IF st_config_achse.b_config_fertig THEN
	(* Fehlermeldungen und Betriebsmeldungen ab dem Startindex in die globalen Meldungsarrays schreiben *)
	garr_stoermeldungen[st_config_achse.i16_meld_startindex + 0] := st_sm.b_achse_nicht_bb;
	garr_stoermeldungen[st_config_achse.i16_meld_startindex + 1] := st_sm.b_achse_nicht_referenziert;
	garr_stoermeldungen[st_config_achse.i16_meld_startindex + 2] := st_sm.b_keine_verfahrfreigabe;
	garr_stoermeldungen[st_config_achse.i16_meld_startindex + 3] := st_sm.b_achse_nicht_auf_startpos;
	garr_stoermeldungen[st_config_achse.i16_meld_startindex + 4] := st_sm.b_ende_skalierungs_nocke;
	garr_stoermeldungen[st_config_achse.i16_meld_startindex + 5] := st_sm.b_ende_camming_nocke;
	garr_stoermeldungen[st_config_achse.i16_meld_startindex + 6] := st_sm.b_skalierung_noch_aktiv;
	garr_stoermeldungen[st_config_achse.i16_meld_startindex + 7] := FALSE;
	garr_stoermeldungen[st_config_achse.i16_meld_startindex + 8] := FALSE;
	garr_stoermeldungen[st_config_achse.i16_meld_startindex + 9] := FALSE;
	garr_stoermeldungen[st_config_achse.i16_meld_startindex + 10] := sm_kein_nocken_definiert;
	garr_stoermeldungen[st_config_achse.i16_meld_startindex + 11] := FALSE;
	garr_stoermeldungen[st_config_achse.i16_meld_startindex + 12] := FALSE;
	garr_stoermeldungen[st_config_achse.i16_meld_startindex + 13] := FALSE;
	garr_stoermeldungen[st_config_achse.i16_meld_startindex + 14] := FALSE;
	garr_stoermeldungen[st_config_achse.i16_meld_startindex + 15] := FALSE;
	garr_stoermeldungen[st_config_achse.i16_meld_startindex + 16] := st_drive_cmd.meldungen.sm_write_soe_parameter;
	garr_stoermeldungen[st_config_achse.i16_meld_startindex + 17] := st_drive_cmd.meldungen.sm_read_soe_parameter;
	garr_stoermeldungen[st_config_achse.i16_meld_startindex + 18] := st_drive_cmd.meldungen.sm_write_nc_parameter;
	garr_stoermeldungen[st_config_achse.i16_meld_startindex + 19] := st_drive_cmd.meldungen.sm_read_nc_parameter;
	garr_stoermeldungen[st_config_achse.i16_meld_startindex + 20] := st_drive_cmd.meldungen.sm_power_enable;
	garr_stoermeldungen[st_config_achse.i16_meld_startindex + 21] := st_drive_cmd.meldungen.sm_power_disable;
	garr_stoermeldungen[st_config_achse.i16_meld_startindex + 22] := st_drive_cmd.meldungen.sm_reset;
	garr_stoermeldungen[st_config_achse.i16_meld_startindex + 23] := st_drive_cmd.meldungen.sm_home;
	garr_stoermeldungen[st_config_achse.i16_meld_startindex + 24] := st_drive_cmd.meldungen.sm_setposition;
	garr_stoermeldungen[st_config_achse.i16_meld_startindex + 25] := st_drive_cmd.meldungen.sm_jog_vorwaerts;
	garr_stoermeldungen[st_config_achse.i16_meld_startindex + 26] := st_drive_cmd.meldungen.sm_jog_rueckwaerts;
	garr_stoermeldungen[st_config_achse.i16_meld_startindex + 27] := st_drive_cmd.meldungen.sm_move_absolute;
	garr_stoermeldungen[st_config_achse.i16_meld_startindex + 28] := st_drive_cmd.meldungen.sm_move_relative;
	garr_stoermeldungen[st_config_achse.i16_meld_startindex + 29] := st_drive_cmd.meldungen.sm_move_velocity;
	garr_stoermeldungen[st_config_achse.i16_meld_startindex + 30] := st_drive_cmd.meldungen.sm_move_modulo;
	garr_stoermeldungen[st_config_achse.i16_meld_startindex + 31] := st_drive_cmd.meldungen.sm_stop_axis;
	garr_stoermeldungen[st_config_achse.i16_meld_startindex + 32] := st_drive_cmd.meldungen.sm_halt_axis;
	garr_stoermeldungen[st_config_achse.i16_meld_startindex + 33] := st_drive_cmd.meldungen.sm_motion_command_timeout;
	garr_stoermeldungen[st_config_achse.i16_meld_startindex + 34] := st_sm.b_achsfehler;
	garr_stoermeldungen[st_config_achse.i16_meld_startindex + 35] := st_sm.b_devicefehler;
	garr_stoermeldungen[st_config_achse.i16_meld_startindex + 36] := st_drive_cmd.meldungen.sm_limit_positiv_erreicht;
	garr_stoermeldungen[st_config_achse.i16_meld_startindex + 37] := st_drive_cmd.meldungen.sm_limit_negativ_erreicht;
	garr_stoermeldungen[st_config_achse.i16_meld_startindex + 38] := st_drive_cmd.meldungen.sm_ec_coe_sdo_write_ex;
	garr_stoermeldungen[st_config_achse.i16_meld_startindex + 39] := st_drive_cmd.meldungen.sm_ec_coe_sdo_read_ex;
	garr_stoermeldungen[st_config_achse.i16_meld_startindex + 40] := FALSE;
	garr_stoermeldungen[st_config_achse.i16_meld_startindex + 41] := FALSE;
	garr_stoermeldungen[st_config_achse.i16_meld_startindex + 42] := FALSE;
	garr_stoermeldungen[st_config_achse.i16_meld_startindex + 43] := FALSE;
	garr_stoermeldungen[st_config_achse.i16_meld_startindex + 44] := FALSE;
	garr_stoermeldungen[st_config_achse.i16_meld_startindex + 45] := FALSE;
	garr_stoermeldungen[st_config_achse.i16_meld_startindex + 46] := FALSE;
	garr_stoermeldungen[st_config_achse.i16_meld_startindex + 47] := FALSE;
	garr_stoermeldungen[st_config_achse.i16_meld_startindex + 48] := FALSE;
	garr_stoermeldungen[st_config_achse.i16_meld_startindex + 49] := FALSE;

	garr_betriebsmeldungen[st_config_achse.i16_meld_startindex + 0] := FALSE;
	garr_betriebsmeldungen[st_config_achse.i16_meld_startindex + 1] := FALSE;
	garr_betriebsmeldungen[st_config_achse.i16_meld_startindex + 2] := FALSE;
	garr_betriebsmeldungen[st_config_achse.i16_meld_startindex + 3] := FALSE;
	garr_betriebsmeldungen[st_config_achse.i16_meld_startindex + 4] := FALSE;
	garr_betriebsmeldungen[st_config_achse.i16_meld_startindex + 5] := FALSE;
	garr_betriebsmeldungen[st_config_achse.i16_meld_startindex + 6] := FALSE;
	garr_betriebsmeldungen[st_config_achse.i16_meld_startindex + 7] := FALSE;
	garr_betriebsmeldungen[st_config_achse.i16_meld_startindex + 8] := FALSE;
	garr_betriebsmeldungen[st_config_achse.i16_meld_startindex + 9] := FALSE;
	garr_betriebsmeldungen[st_config_achse.i16_meld_startindex + 10] := FALSE;
	garr_betriebsmeldungen[st_config_achse.i16_meld_startindex + 11] := FALSE;
	garr_betriebsmeldungen[st_config_achse.i16_meld_startindex + 12] := FALSE;
	garr_betriebsmeldungen[st_config_achse.i16_meld_startindex + 13] := FALSE;
	garr_betriebsmeldungen[st_config_achse.i16_meld_startindex + 14] := FALSE;
	garr_betriebsmeldungen[st_config_achse.i16_meld_startindex + 15] := FALSE;
	garr_betriebsmeldungen[st_config_achse.i16_meld_startindex + 16] := FALSE;
	garr_betriebsmeldungen[st_config_achse.i16_meld_startindex + 17] := FALSE;
	garr_betriebsmeldungen[st_config_achse.i16_meld_startindex + 18] := FALSE;
	garr_betriebsmeldungen[st_config_achse.i16_meld_startindex + 19] := FALSE;
	garr_betriebsmeldungen[st_config_achse.i16_meld_startindex + 20] := FALSE;
	garr_betriebsmeldungen[st_config_achse.i16_meld_startindex + 21] := FALSE;
	garr_betriebsmeldungen[st_config_achse.i16_meld_startindex + 22] := FALSE;
	garr_betriebsmeldungen[st_config_achse.i16_meld_startindex + 23] := FALSE;
	garr_betriebsmeldungen[st_config_achse.i16_meld_startindex + 24] := FALSE;
	garr_betriebsmeldungen[st_config_achse.i16_meld_startindex + 25] := FALSE;
	garr_betriebsmeldungen[st_config_achse.i16_meld_startindex + 26] := FALSE;
	garr_betriebsmeldungen[st_config_achse.i16_meld_startindex + 27] := FALSE;
	garr_betriebsmeldungen[st_config_achse.i16_meld_startindex + 28] := FALSE;
	garr_betriebsmeldungen[st_config_achse.i16_meld_startindex + 29] := FALSE;
	garr_betriebsmeldungen[st_config_achse.i16_meld_startindex + 30] := FALSE;
	garr_betriebsmeldungen[st_config_achse.i16_meld_startindex + 31] := FALSE;
	garr_betriebsmeldungen[st_config_achse.i16_meld_startindex + 32] := FALSE;
	garr_betriebsmeldungen[st_config_achse.i16_meld_startindex + 33] := FALSE;
	garr_betriebsmeldungen[st_config_achse.i16_meld_startindex + 34] := FALSE;
	garr_betriebsmeldungen[st_config_achse.i16_meld_startindex + 35] := FALSE;
	garr_betriebsmeldungen[st_config_achse.i16_meld_startindex + 36] := FALSE;
	garr_betriebsmeldungen[st_config_achse.i16_meld_startindex + 37] := FALSE;
	garr_betriebsmeldungen[st_config_achse.i16_meld_startindex + 38] := FALSE;
	garr_betriebsmeldungen[st_config_achse.i16_meld_startindex + 39] := FALSE;
	garr_betriebsmeldungen[st_config_achse.i16_meld_startindex + 40] := FALSE;
	garr_betriebsmeldungen[st_config_achse.i16_meld_startindex + 41] := FALSE;
	garr_betriebsmeldungen[st_config_achse.i16_meld_startindex + 42] := FALSE;
	garr_betriebsmeldungen[st_config_achse.i16_meld_startindex + 43] := FALSE;
	garr_betriebsmeldungen[st_config_achse.i16_meld_startindex + 44] := FALSE;
	garr_betriebsmeldungen[st_config_achse.i16_meld_startindex + 45] := FALSE;
	garr_betriebsmeldungen[st_config_achse.i16_meld_startindex + 46] := FALSE;
	garr_betriebsmeldungen[st_config_achse.i16_meld_startindex + 47] := FALSE;
	garr_betriebsmeldungen[st_config_achse.i16_meld_startindex + 48] := FALSE;
	garr_betriebsmeldungen[st_config_achse.i16_meld_startindex + 49] := FALSE;
END_IF
END_PROGRAM

(* POU Maschine1720/WT Transport/ST_WT_Transport_Warteposition_1720, ST *)
PROGRAM ST_WT_Transport_Warteposition_1720
VAR_INPUT
	st_config								: struct_config;
	st_ctrl_in								: struct_ctrl_in;
	e_station_vorher_in_anforderung			: BOOL := FALSE;
	e_station_vorher_in_abgegeben			: BOOL := FALSE;
END_VAR
VAR_IN_OUT
	st_visu								: struct_visu;
END_VAR
VAR_OUTPUT
	st_ctrl_out							: struct_ctrl_out;
	a_station_vorher_out_erlaubnis			: BOOL := FALSE;
	a_station_vorher_out_angekommen		: BOOL := FALSE;
END_VAR
VAR
	fb_ton_uez							: TON;
	fb_ton_wz							: TON;
	fb_ton_quitt							: TON;
	fb_ton_wt_auf_wartepos				: TON;
	fb_tof_wt_auf_wartepos					: TOF;
	fb_r_trig_start							: R_TRIG;
	fb_r_trig_wartepos						: R_TRIG;
	fb_r_trig_wartepos_verlassen			: R_TRIG;
	fb_state_entry							: ST_StateEntry;
	sm_wt_hat_wartepos_nicht_verlassen	: BOOL := FALSE;
	sm_wt_hat_wartepos_ueberfahren		: BOOL := FALSE;
	bm_warte_anforderung					: BOOL := FALSE;
	bm_warte_wt_an_stopper				: BOOL := FALSE;
	bm_warte_beladepos_frei				: BOOL := FALSE;

	e_wt_auf_wartepos					AT %I* : BOOL;
	e_wt_wartepos_verlassen				AT %I* : BOOL;
END_VAR
(* Zeiten *)
fb_ton_uez(IN:= , PT:= , Q=>  , ET=> );
fb_ton_wz(IN:= , PT:= , Q=> , ET=> );
fb_ton_quitt(IN:= , PT:= t#100ms, Q=> , ET=> );

fb_ton_wt_auf_wartepos(IN:= e_wt_auf_wartepos, PT:= t#200ms, Q=> , ET=> );
fb_tof_wt_auf_wartepos(IN:= e_wt_auf_wartepos, PT:= t#200ms, Q=> , ET=> );

(* Flanken *)
fb_r_trig_wartepos(CLK:= e_wt_auf_wartepos, Q=> );
fb_r_trig_wartepos_verlassen(CLK:= e_wt_wartepos_verlassen, Q=> );
fb_r_trig_start(CLK:= st_ctrl_in.b_start, Q=> );

(* ==================================Toplevel=================================== *)
IF fb_state_entry.i16_next_step > INIT AND fb_state_entry.i16_next_step < FEHLER THEN
	(* Allgemeine Fehler *)
	IF st_ctrl_in.b_stop THEN
		fb_state_entry.i16_next_step := STOP;
	ELSIF zyl_wt_stopper_einlauf.st_ctrl.out.b_fehler THEN
		fb_state_entry.i16_next_step := FEHLER;
	(* Zylinder im Handbetrieb *)
	ELSIF gi16_betriebsart = HAND AND
		st_visu.st_zyl.i16_nr_zyl_im_handbetrieb = zyl_wt_stopper_einlauf.fb.st_config.i16_identnummer
		THEN
			fb_state_entry.i16_next_step := FEHLER;
	END_IF
END_IF

(* ============================Haupt-Schrittkette================================ *)
fb_state_entry(
	i16_next_step:= , 
	i16_pos:= 1,
	s_debugtext:= ,
	E=> ,
	X=> , 
	i16_step=> ,
	i16_last_step=> );

CASE fb_state_entry.i16_step OF
(*=======================================================*)
	INIT_OBJ:
		IF st_config.b_config_fertig THEN
			fb_state_entry.i16_next_step := INIT;
		END_IF

(*=======================================================*)
	INIT:
		IF fb_state_entry.E THEN
			fb_ton_wz.IN := FALSE;
			fb_ton_uez.IN := FALSE;
			fb_ton_quitt.IN := FALSE;
			st_ctrl_out.b_fehler := FALSE;
			st_ctrl_out.b_bereit := FALSE;
			st_ctrl_out.b_fertig := FALSE;
			st_ctrl_out.b_kontroller_start := FALSE;
			zyl_wt_stopper_einlauf.st_ctrl.in.b_einfahren := FALSE;
			zyl_wt_stopper_einlauf.st_ctrl.in.b_ausfahren := FALSE;
			sm_wt_hat_wartepos_nicht_verlassen := FALSE;
			sm_wt_hat_wartepos_ueberfahren := FALSE;
			bm_warte_anforderung := FALSE;
			bm_warte_wt_an_stopper := FALSE;
			bm_warte_beladepos_frei := FALSE;
			a_station_vorher_out_erlaubnis := FALSE;
			a_station_vorher_out_angekommen := FALSE;
		END_IF

		(*-----------------------Weiterschaltbedingungen----------------------------*)
		IF st_ctrl_in.b_init THEN
			zyl_wt_stopper_einlauf.st_ctrl.in.b_quittieren := FALSE;
			fb_state_entry.i16_next_step := 20;
		END_IF

(*=======================================================*)
	20: (* Initialisierung: Einlaufstopper ausfahren *)
		IF fb_state_entry.E THEN
			zyl_wt_stopper_einlauf.st_ctrl.in.b_ausfahren := TRUE;
		END_IF

		(*-----------------------Weiterschaltbedingungen----------------------------*)
		IF zyl_wt_stopper_einlauf.st_ctrl.out.b_ausgefahren THEN
			zyl_wt_stopper_einlauf.st_ctrl.in.b_ausfahren := FALSE;
			fb_state_entry.i16_next_step :=  BEREIT;
		END_IF

(*=======================================================*)
	BEREIT:	(* Warte auf Start von Kontroller *)
		IF fb_state_entry.E THEN
			st_ctrl_out.b_bereit := TRUE;
			st_ctrl_out.b_fertig := TRUE;
		END_IF

	(*-----------------------Weiterschaltbedingungen----------------------------*)
		IF st_config.b_station_aktiv OR st_config.b_station_in_simulation THEN
			(* WT Transport aktiv oder in Simulation *)
			IF st_ctrl_in.b_start THEN
			(* WT Transport gestartet *)
				st_ctrl_out.b_fertig := FALSE;
				fb_state_entry.i16_next_step := 110;
			END_IF
		ELSE
			fb_state_entry.i16_next_step := 500;
		END_IF

(*=======================================================*)
	110: (* Statische WT-Abfrage auf Warteposition nach der Initialisierung *)
		IF fb_state_entry.E THEN
			st_ctrl_out.b_kontroller_start := TRUE;
		END_IF

		IF NOT e_station_vorher_in_abgegeben THEN
			a_station_vorher_out_angekommen := FALSE;
		END_IF

		(*-----------------------Weiterschaltbedingungen----------------------------*)
		IF e_wt_auf_wartepos THEN
			st_ctrl_out.b_kontroller_start := FALSE;
			fb_state_entry.i16_next_step := 140;
		ELSE	(* Kein WT da, deshalb einen holen *)
			st_ctrl_out.b_kontroller_start := FALSE;
			fb_state_entry.i16_next_step := 120;
		END_IF

(*=======================================================*)
	120: (* Kein WT da -> warte auf Anforderung von vorheriger Station *)
		IF fb_state_entry.E THEN
			st_ctrl_out.b_kontroller_start := TRUE;
			bm_warte_anforderung := TRUE;
		END_IF

		IF NOT e_station_vorher_in_abgegeben THEN
			a_station_vorher_out_angekommen := FALSE;
		END_IF

		(*-----------------------Weiterschaltbedingungen----------------------------*)
		IF e_station_vorher_in_anforderung THEN
			a_station_vorher_out_angekommen := FALSE;
			a_station_vorher_out_erlaubnis := TRUE;
			st_ctrl_out.b_kontroller_start := FALSE;
			bm_warte_anforderung := FALSE;
			fb_state_entry.i16_next_step := 130;
		END_IF

(*=======================================================*)
	130: (* Warte bis WT an Stopper angekommen ist *)
		IF fb_state_entry.E THEN
			st_ctrl_out.b_kontroller_start := TRUE;
			bm_warte_wt_an_stopper := TRUE;
		END_IF

		(*-----------------------Weiterschaltbedingungen----------------------------*)
		IF fb_r_trig_wartepos.Q THEN
			a_station_vorher_out_erlaubnis := FALSE;
			a_station_vorher_out_angekommen := TRUE;
			st_ctrl_out.b_kontroller_start := FALSE;
			fb_ton_uez.IN := FALSE;
			bm_warte_wt_an_stopper := FALSE;
			fb_state_entry.i16_next_step := 140;
		END_IF

(*=======================================================*)
	140: (* WT ist da - Warten bis Beladeposition auf Bestücktisch frei ist *)
		IF fb_state_entry.E THEN
			zyl_wt_stopper_einlauf.st_ctrl.in.b_ausfahren := FALSE;
			zyl_wt_stopper_einlauf.st_ctrl.in.b_einfahren := FALSE;
			bm_warte_beladepos_frei := TRUE;
		END_IF

		(*-----------------------Weiterschaltbedingungen----------------------------*)
		IF NOT ST_WT_Transport_Beladen_1720.e_wt_auf_beladepos AND NOT axis_z_achse.st_ctrl.in.b_start THEN
			bm_warte_beladepos_frei := FALSE;
			fb_state_entry.i16_next_step := 150;
		ELSIF e_wt_wartepos_verlassen THEN
			(* Warteposition wurde unerlaubterweise überfahren *)
			sm_wt_hat_wartepos_ueberfahren := TRUE;
			fb_state_entry.i16_next_step := FEHLER;
		END_IF

(*=======================================================*)
	150: (* Bestücktisch ist frei -> Einlaufstopper einfahren *)
		IF fb_state_entry.E THEN
			zyl_wt_stopper_einlauf.st_ctrl.in.b_einfahren := TRUE;
		END_IF

		(*-----------------------Weiterschaltbedingungen----------------------------*)
		IF zyl_wt_stopper_einlauf.st_ctrl.out.b_eingefahren THEN
			zyl_wt_stopper_einlauf.st_ctrl.in.b_einfahren := FALSE;
			fb_state_entry.i16_next_step := 160;
		END_IF

(*=======================================================*)
	160: (* WT fährt weiter - Überwachung starten *)
		IF fb_state_entry.E THEN
			fb_ton_uez.PT := t#5s;
 			fb_ton_uez.IN := TRUE;
			st_ctrl_out.b_kontroller_start := TRUE;
		END_IF

		(*-----------------------Weiterschaltbedingungen----------------------------*)
		IF fb_r_trig_wartepos_verlassen.Q THEN
			fb_ton_uez.IN := FALSE;
			st_ctrl_out.b_kontroller_start := FALSE;
			fb_state_entry.i16_next_step := 170;
		ELSIF fb_ton_uez.Q THEN
			sm_wt_hat_wartepos_nicht_verlassen := TRUE;
			fb_state_entry.i16_next_step := FEHLER;
		END_IF

(*=======================================================*)
	170: (* Einlaufstopper ausfahren *)
		IF fb_state_entry.E THEN
			fb_ton_wz.IN := TRUE;
			fb_ton_wz.PT := t#1s;
			zyl_wt_stopper_einlauf.st_ctrl.in.b_ausfahren := TRUE;
		END_IF

		(*-----------------------Weiterschaltbedingungen----------------------------*)
		IF zyl_wt_stopper_einlauf.st_ctrl.out.b_ausgefahren AND fb_ton_wz.Q THEN
			zyl_wt_stopper_einlauf.st_ctrl.in.b_ausfahren := FALSE;
			fb_state_entry.i16_next_step := BEREIT;
			fb_ton_wz.IN := FALSE;
		END_IF

(*=======================================================*)
	500: (* Einlaufstopper einfahren, damit WTs auf Bestücktisch geschoben werden können. *)
		IF fb_state_entry.E THEN
			zyl_wt_stopper_einlauf.st_ctrl.in.b_einfahren := TRUE;
		END_IF

		(*-----------------------Weiterschaltbedingungen----------------------------*)
		IF zyl_wt_stopper_einlauf.st_ctrl.out.b_eingefahren THEN
			zyl_wt_stopper_einlauf.st_ctrl.in.b_einfahren := FALSE;
			fb_state_entry.i16_next_step :=  510;
		END_IF

(*=======================================================*)
	510:	(* Warte auf Konfigurationsänderung *)

	(*-----------------------Weiterschaltbedingungen----------------------------*)
		IF st_config.b_station_aktiv OR st_config.b_station_in_simulation THEN
			(* WT Transport aktiv oder in Simulation *)
			fb_state_entry.i16_next_step := BEREIT;
		END_IF

(*=======================================================*)
	FEHLER:
		IF fb_state_entry.E THEN
			st_ctrl_out.b_fehler := TRUE;
			fb_ton_quitt.IN := FALSE;
			zyl_wt_stopper_einlauf.st_ctrl.in.b_quittieren := FALSE;

			a_station_vorher_out_erlaubnis := FALSE;
			a_station_vorher_out_angekommen := FALSE;
		END_IF

		(*-----------------------Weiterschaltbedingungen----------------------------*)
		IF st_ctrl_in.b_quitt AND NOT fb_state_entry.E THEN
			st_ctrl_out.b_fehler := FALSE;
			zyl_wt_stopper_einlauf.st_ctrl.in.b_quittieren := TRUE;
			fb_ton_quitt.IN := TRUE;
		END_IF

		IF fb_ton_quitt.Q THEN
			fb_ton_quitt.IN := FALSE;
			fb_state_entry.i16_next_step := INIT;
		END_IF

(*=======================================================*)
	STOP:
		IF fb_state_entry.E THEN
			fb_ton_quitt.IN := FALSE;
			st_ctrl_out.b_kontroller_start := FALSE;
			zyl_wt_stopper_einlauf.st_ctrl.in.b_quittieren := FALSE;
			a_station_vorher_out_erlaubnis := FALSE;
			a_station_vorher_out_angekommen := FALSE;
		END_IF

		(*-----------------------Weiterschaltbedingungen----------------------------*)
		IF st_ctrl_in.b_quitt AND NOT fb_state_entry.E THEN
			fb_ton_quitt.IN := TRUE;
			zyl_wt_stopper_einlauf.st_ctrl.in.b_quittieren := TRUE;
		END_IF

		IF fb_ton_quitt.Q THEN
			fb_ton_quitt.IN := FALSE;
			fb_state_entry.i16_next_step := INIT;
		END_IF
END_CASE

fb_state_entry(
	i16_next_step:= ,
	i16_pos:= 2,
	s_debugtext:= ,
	E=> ,
	X=> ,
	i16_step=> ,
	i16_last_step=> );

IF st_config.b_config_fertig THEN
	(* Fehlermeldungen ab dem Startindex in das globale Störmeldungsarray schreiben *)
	garr_stoermeldungen[st_config.i16_meld_startindex + 0] := sm_wt_hat_wartepos_nicht_verlassen;
	garr_stoermeldungen[st_config.i16_meld_startindex + 1] := sm_wt_hat_wartepos_ueberfahren;
	garr_stoermeldungen[st_config.i16_meld_startindex + 2] := FALSE;
	garr_stoermeldungen[st_config.i16_meld_startindex + 3] := FALSE;
	garr_stoermeldungen[st_config.i16_meld_startindex + 4] := FALSE;
	garr_stoermeldungen[st_config.i16_meld_startindex + 5] := FALSE;
	garr_stoermeldungen[st_config.i16_meld_startindex + 6] := FALSE;
	garr_stoermeldungen[st_config.i16_meld_startindex + 7] := FALSE;
	garr_stoermeldungen[st_config.i16_meld_startindex + 8] := FALSE;
	garr_stoermeldungen[st_config.i16_meld_startindex + 9] := FALSE;
	garr_stoermeldungen[st_config.i16_meld_startindex + 10] := FALSE;
	garr_stoermeldungen[st_config.i16_meld_startindex + 11] := FALSE;
	garr_stoermeldungen[st_config.i16_meld_startindex + 12] := FALSE;
	garr_stoermeldungen[st_config.i16_meld_startindex + 13] := FALSE;
	garr_stoermeldungen[st_config.i16_meld_startindex + 14] := FALSE;
	garr_stoermeldungen[st_config.i16_meld_startindex + 15] := FALSE;
	garr_stoermeldungen[st_config.i16_meld_startindex + 16] := FALSE;
	garr_stoermeldungen[st_config.i16_meld_startindex + 17] := FALSE;
	garr_stoermeldungen[st_config.i16_meld_startindex + 18] := FALSE;
	garr_stoermeldungen[st_config.i16_meld_startindex + 19] := FALSE;
	
	garr_betriebsmeldungen[st_config.i16_meld_startindex + 0] := bm_warte_anforderung;
	garr_betriebsmeldungen[st_config.i16_meld_startindex + 1] := bm_warte_wt_an_stopper;
	garr_betriebsmeldungen[st_config.i16_meld_startindex + 2] := bm_warte_beladepos_frei;
	garr_betriebsmeldungen[st_config.i16_meld_startindex + 3] := FALSE;
	garr_betriebsmeldungen[st_config.i16_meld_startindex + 4] := FALSE;
	garr_betriebsmeldungen[st_config.i16_meld_startindex + 5] := FALSE;
	garr_betriebsmeldungen[st_config.i16_meld_startindex + 6] := FALSE;
	garr_betriebsmeldungen[st_config.i16_meld_startindex + 7] := FALSE;
	garr_betriebsmeldungen[st_config.i16_meld_startindex + 8] := FALSE;
	garr_betriebsmeldungen[st_config.i16_meld_startindex + 9] := FALSE;
	garr_betriebsmeldungen[st_config.i16_meld_startindex + 10] := FALSE;
	garr_betriebsmeldungen[st_config.i16_meld_startindex + 11] := FALSE;
	garr_betriebsmeldungen[st_config.i16_meld_startindex + 12] := FALSE;
	garr_betriebsmeldungen[st_config.i16_meld_startindex + 13] := FALSE;
	garr_betriebsmeldungen[st_config.i16_meld_startindex + 14] := FALSE;
	garr_betriebsmeldungen[st_config.i16_meld_startindex + 15] := FALSE;
	garr_betriebsmeldungen[st_config.i16_meld_startindex + 16] := FALSE;
	garr_betriebsmeldungen[st_config.i16_meld_startindex + 17] := FALSE;
	garr_betriebsmeldungen[st_config.i16_meld_startindex + 18] := FALSE;
	garr_betriebsmeldungen[st_config.i16_meld_startindex + 19] := FALSE;
END_IF
END_PROGRAM

(* POU EPT Lib/Funktionen/DT_TO_SPECIALSTRING_YYYY_MM, ST *)
FUNCTION DT_TO_SPECIALSTRING_YYYY_MM : STRING
VAR_INPUT
	inDT					:	DT;
END_VAR
VAR

	TempString		:	STRING;
	SysTime				:	TIMESTRUCT;


	wYear					: WORD;
	wMonth				: WORD;
	wDay					: WORD;
	wHour					: WORD;
	wMin					: WORD;
	wSec					: WORD;
END_VAR
(*gVarStrSystemTime:=SYSTEMTIME_TO_STRING(gFB_GETLOCALSYSTEMTIME.systemTime);
gVarDTSystemtime:=SYSTEMTIME_TO_DT(gFB_GETLOCALSYSTEMTIME.SystemTime);
gVarSystemtime:=gFB_GETLOCALSYSTEMTIME.systemTime;
*)

SysTime:=DT_TO_SYSTEMTIME(inDT);

wYear:=SysTime.wYear;
wMonth:=SysTime.wMonth;
wDay:=SysTime.wDay;
wHour:=SysTime.wHour;
wMin:=SysTime.wMinute;
wSec:=SysTime.wSecond;
TempString:='';

TempString:=CONCAT(TempString ,WORD_TO_STRING(wYear));
TempString:=CONCAT(TempString ,'_');

IF wMonth<10 THEN	TempString:=CONCAT(TempString ,WORD_TO_STRING(0)); END_IF;
TempString:=CONCAT(TempString ,WORD_TO_STRING(wMonth));


DT_TO_SPECIALSTRING_YYYY_MM:=TempString;
END_FUNCTION

(* POU Gemeinsamkeiten17xx/Initialisierung/Startup/ST_Datainit_Achsen, ST *)
PROGRAM ST_Datainit_Achsen
VAR
	b_config_fertig			: BOOL := FALSE;
END_VAR
IF	NOT axis_bestueckachse.st_config.b_config_fertig OR
	NOT axis_virt_master.st_config.b_config_fertig OR
	NOT axis_z_achse.st_config.b_config_fertig OR
	NOT axis_y_achse.st_config.b_config_fertig OR
	NOT axis_bandeinzug_achse.st_config.b_config_fertig OR
	NOT axis_transport_wt_achse.st_config.b_config_fertig
	THEN
		CASE gst_datensatz.st_md.i16_typ_zelle OF
			KEINE_ZELLE:
				;
			BESTUECKZELLE_1700:
				(* Virtuelle Masterachse *)
				axis_virt_master.st_config.b_config_fertig := FALSE;
				axis_virt_master.st_config.b_limitsensor_negativ_vorhanden := FALSE;
				axis_virt_master.st_config.b_limitsensor_positiv_vorhanden := FALSE;
				axis_virt_master.st_config.b_refsensor_vorhanden := FALSE;
				axis_virt_master.st_config.r_getriebefaktor := 1.0;
				axis_virt_master.st_config.i16_achstyp := RUND_VIRTUELL;
				axis_virt_master.st_config.i16_meld_startindex := 1400;
				axis_virt_master.st_config.s_beschreibung := ' ';
				axis_virt_master.st_config.s_instanz_name := 'Virtuelle Masterachse';
				axis_virt_master.st_config.ui16_ethercat_slave_id := 0;
				axis_virt_master.st_config.ui16_ethercat_adr := 0;
				axis_virt_master.st_config.b_config_fertig := TRUE;
				(* Bestueckachse *)
				axis_bestueckachse.st_config.b_config_fertig := FALSE;
				axis_bestueckachse.st_config.b_limitsensor_negativ_vorhanden := FALSE;
				axis_bestueckachse.st_config.b_limitsensor_positiv_vorhanden := FALSE;
				axis_bestueckachse.st_config.b_refsensor_vorhanden := FALSE;
				axis_bestueckachse.st_config.r_getriebefaktor := 1.0;
				axis_bestueckachse.st_config.i16_achstyp := RUND;
				axis_bestueckachse.st_config.i16_meld_startindex := 1000;
				axis_bestueckachse.st_config.s_beschreibung := ' ';
				axis_bestueckachse.st_config.s_instanz_name := 'Bestückachse';
				axis_bestueckachse.st_config.ui16_ethercat_slave_id := 42;
				axis_bestueckachse.st_config.ui16_ethercat_adr := 1024;
				axis_bestueckachse.st_config.b_config_fertig := TRUE;
				(* Servobandeinzug *)
				axis_bandeinzug_achse.st_config.b_config_fertig := FALSE;
				axis_bandeinzug_achse.st_config.b_limitsensor_negativ_vorhanden := FALSE;
				axis_bandeinzug_achse.st_config.b_limitsensor_positiv_vorhanden := FALSE;
				axis_bandeinzug_achse.st_config.b_refsensor_vorhanden := FALSE;
				axis_bandeinzug_achse.st_config.r_getriebefaktor := 1.0;
				axis_bandeinzug_achse.st_config.i16_achstyp := RUND;
				axis_bandeinzug_achse.st_config.i16_meld_startindex := 1300;
				axis_bandeinzug_achse.st_config.s_beschreibung := ' ';
				axis_bandeinzug_achse.st_config.s_instanz_name := 'Servobandeinzug';
				axis_bandeinzug_achse.st_config.ui16_ethercat_slave_id := 42;
				axis_bandeinzug_achse.st_config.ui16_ethercat_adr := 1024;
				(* Z-Achse *)
				axis_z_achse.st_config.b_config_fertig := FALSE;
				axis_z_achse.st_config.b_limitsensor_negativ_vorhanden := FALSE;
				axis_z_achse.st_config.b_limitsensor_positiv_vorhanden := FALSE;
				axis_z_achse.st_config.b_refsensor_vorhanden := FALSE;
				axis_z_achse.st_config.r_getriebefaktor := 1.0;
				axis_z_achse.st_config.i16_achstyp := LINEAR;
				axis_z_achse.st_config.i16_meld_startindex := 1100;
				axis_z_achse.st_config.s_beschreibung := ' ';
				axis_z_achse.st_config.s_instanz_name := 'Z-Achse';
				axis_z_achse.st_config.ui16_ethercat_slave_id := 43;
				axis_z_achse.st_config.ui16_ethercat_adr := 1026;
				axis_z_achse.st_config.b_config_fertig := TRUE;
				(* Y-Achse *)
				axis_y_achse.st_config.b_config_fertig := FALSE;
				axis_y_achse.st_config.b_limitsensor_negativ_vorhanden := FALSE;
				axis_y_achse.st_config.b_limitsensor_positiv_vorhanden := FALSE;
				axis_y_achse.st_config.b_refsensor_vorhanden := FALSE;
				axis_y_achse.st_config.r_getriebefaktor := 1.0;
				axis_y_achse.st_config.i16_achstyp := LINEAR;
				axis_y_achse.st_config.i16_meld_startindex := 1200;
				axis_y_achse.st_config.s_beschreibung := ' ';
				axis_y_achse.st_config.s_instanz_name := 'Y-Achse';
				axis_y_achse.st_config.ui16_ethercat_slave_id := 43;
				axis_y_achse.st_config.ui16_ethercat_adr := 1026;
				axis_y_achse.st_config.b_config_fertig := TRUE;
				(* Transport WT Achse *)
				axis_transport_wt_achse.st_config.b_config_fertig := FALSE;
				axis_transport_wt_achse.st_config.b_limitsensor_negativ_vorhanden := FALSE;
				axis_transport_wt_achse.st_config.b_limitsensor_positiv_vorhanden := FALSE;
				axis_transport_wt_achse.st_config.b_refsensor_vorhanden := FALSE;
				axis_transport_wt_achse.st_config.r_getriebefaktor := 1.0;
				axis_transport_wt_achse.st_config.i16_achstyp := LINEAR;
				axis_transport_wt_achse.st_config.i16_meld_startindex := 1500;
				axis_transport_wt_achse.st_config.s_beschreibung := ' ';
				axis_transport_wt_achse.st_config.s_instanz_name := 'Transport_WT_Achse';
				axis_transport_wt_achse.st_config.ui16_ethercat_slave_id :=43;
				axis_transport_wt_achse.st_config.ui16_ethercat_adr :=1026;
				axis_transport_wt_achse.st_config.b_config_fertig := TRUE;

				axis_bandeinzug_achse.st_config.b_config_fertig := TRUE;

			BESTUECKZELLE_1720:
				(* Virtuelle Masterachse *)
				axis_virt_master.st_config.b_config_fertig := FALSE;
				axis_virt_master.st_config.b_limitsensor_negativ_vorhanden := FALSE;
				axis_virt_master.st_config.b_limitsensor_positiv_vorhanden := FALSE;
				axis_virt_master.st_config.b_refsensor_vorhanden := FALSE;
				axis_virt_master.st_config.r_getriebefaktor := 1.0;
				axis_virt_master.st_config.i16_achstyp := RUND_VIRTUELL;
				axis_virt_master.st_config.i16_meld_startindex := 1400;
				axis_virt_master.st_config.s_beschreibung := ' ';
				axis_virt_master.st_config.s_instanz_name := 'Virtuelle Masterachse';
				axis_virt_master.st_config.ui16_ethercat_slave_id := 0;
				axis_virt_master.st_config.ui16_ethercat_adr := 0;
				axis_virt_master.st_config.b_config_fertig := TRUE;
				(* Bestueckachse *)
				axis_bestueckachse.st_config.b_config_fertig := FALSE;
				axis_bestueckachse.st_config.b_limitsensor_negativ_vorhanden := FALSE;
				axis_bestueckachse.st_config.b_limitsensor_positiv_vorhanden := FALSE;
				axis_bestueckachse.st_config.b_refsensor_vorhanden := FALSE;
				axis_bestueckachse.st_config.r_getriebefaktor := 1.0;
				axis_bestueckachse.st_config.i16_achstyp := RUND;
				axis_bestueckachse.st_config.i16_meld_startindex := 1000;
				axis_bestueckachse.st_config.s_beschreibung := ' ';
				axis_bestueckachse.st_config.s_instanz_name := 'Bestückachse';
				axis_bestueckachse.st_config.ui16_ethercat_slave_id := 40;
				axis_bestueckachse.st_config.ui16_ethercat_adr := 1010;
				axis_bestueckachse.st_config.b_config_fertig := TRUE;
				(* Z-Achse *)
				axis_z_achse.st_config.b_config_fertig := FALSE;
				axis_z_achse.st_config.b_limitsensor_negativ_vorhanden := TRUE;
				axis_z_achse.st_config.b_limitsensor_positiv_vorhanden := TRUE;
				axis_z_achse.st_config.b_refsensor_vorhanden := FALSE;
				axis_z_achse.st_config.r_getriebefaktor := 1.0;
				axis_z_achse.st_config.i16_achstyp := LINEAR;
				axis_z_achse.st_config.i16_meld_startindex := 1100;
				axis_z_achse.st_config.s_beschreibung := ' ';
				axis_z_achse.st_config.s_instanz_name := 'Z-Achse';
				axis_z_achse.st_config.ui16_ethercat_slave_id := 7;
				axis_z_achse.st_config.ui16_ethercat_adr := 1012;
				axis_z_achse.st_config.b_config_fertig := TRUE;

			RASTERFOLIE:
				(* Virtuelle Masterachse *)
				axis_virt_master.st_config.b_config_fertig := FALSE;
				axis_virt_master.st_config.b_limitsensor_negativ_vorhanden := FALSE;
				axis_virt_master.st_config.b_limitsensor_positiv_vorhanden := FALSE;
				axis_virt_master.st_config.b_refsensor_vorhanden := FALSE;
				axis_virt_master.st_config.r_getriebefaktor := 1.0;
				axis_virt_master.st_config.i16_achstyp := RUND_VIRTUELL;
				axis_virt_master.st_config.i16_meld_startindex := 1400;
				axis_virt_master.st_config.s_beschreibung := ' ';
				axis_virt_master.st_config.s_instanz_name := 'Virtuelle Masterachse';
				axis_virt_master.st_config.ui16_ethercat_slave_id := 0;
				axis_virt_master.st_config.ui16_ethercat_adr := 0;
				axis_virt_master.st_config.b_config_fertig := TRUE;
				(* Bestueckachse *)
				axis_bestueckachse.st_config.b_config_fertig := FALSE;
				axis_bestueckachse.st_config.b_limitsensor_negativ_vorhanden := FALSE;
				axis_bestueckachse.st_config.b_limitsensor_positiv_vorhanden := FALSE;
				axis_bestueckachse.st_config.b_refsensor_vorhanden := FALSE;
				axis_bestueckachse.st_config.r_getriebefaktor := 1.0;
				axis_bestueckachse.st_config.i16_achstyp := RUND;
				axis_bestueckachse.st_config.i16_meld_startindex := 1000;
				axis_bestueckachse.st_config.s_beschreibung := ' ';
				axis_bestueckachse.st_config.s_instanz_name := 'Bestückachse';
				axis_bestueckachse.st_config.ui16_ethercat_slave_id := 2;
				axis_bestueckachse.st_config.ui16_ethercat_adr := 1010;
				axis_bestueckachse.st_config.b_config_fertig := TRUE;
				(* Z-Achse *)
				axis_z_achse.st_config.b_config_fertig := FALSE;
				axis_z_achse.st_config.b_limitsensor_negativ_vorhanden := TRUE;
				axis_z_achse.st_config.b_limitsensor_positiv_vorhanden := TRUE;
				axis_z_achse.st_config.b_refsensor_vorhanden := FALSE;
				axis_z_achse.st_config.r_getriebefaktor := 1.0;
				axis_z_achse.st_config.i16_achstyp := LINEAR;
				axis_z_achse.st_config.i16_meld_startindex := 1100;
				axis_z_achse.st_config.s_beschreibung := ' ';
				axis_z_achse.st_config.s_instanz_name := 'Z-Achse';
				axis_z_achse.st_config.ui16_ethercat_slave_id := 2;
				axis_z_achse.st_config.ui16_ethercat_adr := 1012;
				axis_z_achse.st_config.b_config_fertig := TRUE;
				(* Y-Achse *)
				axis_y_achse.st_config.b_config_fertig := FALSE;
				axis_y_achse.st_config.b_limitsensor_negativ_vorhanden := TRUE;
				axis_y_achse.st_config.b_limitsensor_positiv_vorhanden := TRUE;
				axis_y_achse.st_config.b_refsensor_vorhanden := FALSE;
				axis_y_achse.st_config.r_getriebefaktor := 1.0;
				axis_y_achse.st_config.i16_achstyp := LINEAR;
				axis_y_achse.st_config.i16_meld_startindex := 1200;
				axis_y_achse.st_config.s_beschreibung := ' ';
				axis_y_achse.st_config.s_instanz_name := 'Y-Achse';
				axis_y_achse.st_config.ui16_ethercat_slave_id := 2;
				axis_y_achse.st_config.ui16_ethercat_adr := 1012;
				axis_y_achse.st_config.b_config_fertig := TRUE;

		END_CASE
ELSE
	b_config_fertig := TRUE;
END_IF
END_PROGRAM

(* POU EPT Lib/Programmbausteine/ST_UPS, ST *)
PROGRAM ST_UPS
VAR_INPUT
	st_config				: struct_config;
	st_ctrl_in				: struct_ctrl_in;
	b_Ups					: BOOL;
END_VAR
VAR_IN_OUT

END_VAR
VAR_OUTPUT
	st_ctrl_out			: struct_ctrl_out;
END_VAR
VAR
	fb_ton_quitt			: TON;
	fb_ton_uez			: TON;
	fb_state_entry			: ST_StateEntry;

	nLastErrID			:UDINT;

	fbGetUpsStatus		: FB_GetUPSStatus;

	bm_ReplaceBattery 	: BOOL;
	bm_NoPower 		: BOOL;
	bm_StatusNotValid 	: BOOL;
END_VAR
(*======================================================
   ST: ST_UPS
 ------------------------------------------------------
   Auth: 	Thomas Vilgis    						 
   Date: 	21.06.2018    						     
   Rev.: 		1.0	
   Desc:		Der Baustein liest den Status des Akkupacks aus.
			Die restliche Akkulaufzeit in Minuten kann abgefragt werden.
			Wenn der Akkupack getauscht werden muss wird angezeigt.
			Wenn sich der PC im Netzbetrieb befindet wird angezeigt.
   Historie: 	1.0

 ========================================================*)

(* Zeiten *)
fb_ton_quitt(IN:= , PT:= t#100ms, Q=> , ET=> );
fb_ton_uez(IN:= , PT:= t#20s, Q=> , ET=> );

(* Flanken *)


(* Toplevel *)
IF fb_state_entry.i16_next_step > INIT AND fb_state_entry.i16_next_step < FEHLER  THEN
	IF fb_state_entry.i16_next_step < STOP THEN
		IF st_ctrl_in.b_stop THEN
			fb_state_entry.i16_next_step := STOP;
		END_IF
	END_IF
END_IF

(* ======================================Schrittkette======================================== *)
fb_state_entry(	i16_pos:= 1);

CASE fb_state_entry.i16_step OF
(*=======================================================*)
	INIT_OBJ:
		IF st_config.b_config_fertig THEN
			fb_state_entry.i16_next_step := INIT;
		END_IF

(*=======================================================*)
	INIT:
		IF fb_state_entry.E THEN
			fb_ton_quitt.IN := FALSE;
			fb_ton_uez.IN := FALSE;
			st_ctrl_out.b_fehler := FALSE;
			st_ctrl_out.b_bereit := FALSE;
			st_ctrl_out.b_fertig := FALSE;
			st_ctrl_out.b_busy := FALSE;

			bm_ReplaceBattery := FALSE;
			bm_NoPower := FALSE;
			bm_StatusNotValid := FALSE;

			fbGetUpsStatus.bEnable := FALSE;
		END_IF

		(*-----------------------Weiterschaltbedingungen----------------------------*)
		fb_state_entry.i16_next_step := BEREIT;

(*=======================================================*)
	BEREIT:
		IF fb_state_entry.E THEN
			st_ctrl_out.b_bereit := TRUE;
		END_IF

		fbGetUpsStatus.bEnable := b_Ups;
		fb_ton_uez.IN := b_Ups;

		(*-----------------------Weiterschaltbedingungen----------------------------*)
		IF b_Ups THEN
			IF fbGetUpsStatus.bValid THEN
				fb_state_entry.i16_next_step := 110;
			ELSIF fb_ton_uez.Q THEN
				bm_StatusNotValid := TRUE;
				fb_state_entry.i16_next_step := FEHLER;
			END_IF
		END_IF

		IF fb_state_entry.X THEN
			st_ctrl_out.b_bereit := FALSE;
			st_ctrl_out.b_fertig := FALSE;
			st_ctrl_out.b_busy := TRUE;
		END_IF

(*=======================================================*)
	110:	(* Evaluation *)

		(*-----------------------Weiterschaltbedingungen----------------------------*)
		IF fbGetUpsStatus.bValid THEN
			IF NOT fbGetUpsStatus.bError THEN
				CASE fbGetUpsStatus.stStatus.eBatteryStatus OF
					BatteryUnknownStatus:	(*Der Akkustatus ist unbekannt*)
						;
					BatteryOk:			(*Der Akku ist in Ordnung*)
						bm_ReplaceBattery := FALSE;
					BatteryReplace:		(*Der Akku sollte gewechselt werden*)
						bm_ReplaceBattery := TRUE;
				END_CASE

				CASE fbGetUpsStatus.stStatus.eCommStatus OF
					UpsCommUnknownStatus:	(*Kommunikationsstatus zur USV-Hardware ist unbekannt*)
						;
					UpsCommOk:		(*Kommunikation zur USV-Hardware ist hergestellt*)
						;
					UpsCommFailed:	(*Kommunikation zur USV wurde unterbrochen*)
						;
				END_CASE

				CASE fbGetUpsStatus.stStatus.ePowerStatus OF
					PowerUnknownStatus:	(*Der Status der Stromversorgung ist unbekannt*)
						;
					PowerOnLine:		(*Das Gerät befindet sich im Netzbetrieb*)
						bm_NoPower := FALSE;
					PowerOnBattery:	(*Stromausfall ist aufgetreten und das Gerät befindet sich im Akkubetrieb*)
						bm_NoPower := TRUE;
				END_CASE
			ELSE
				nLastErrID := fbGetUpsStatus.nErrId;
				fb_state_entry.i16_next_step := FEHLER;
			END_IF
		ELSE
			bm_StatusNotValid := TRUE;
			fb_state_entry.i16_next_step := FEHLER;
		END_IF

(*=======================================================*)
	STOP, FEHLER:
		IF fb_state_entry.E THEN
			st_ctrl_out.b_fehler := fb_state_entry.i16_step = FEHLER;
			st_ctrl_out.b_gestoppt := fb_state_entry.i16_step = STOP;
			fb_ton_quitt.IN := FALSE;
			fbGetUpsStatus.bEnable := FALSE;
		END_IF

		(*-----------------------Weiterschaltbedingungen----------------------------*)
		IF st_ctrl_in.b_quitt THEN
			st_ctrl_out.b_fehler := FALSE;
			fb_ton_quitt.IN := TRUE;
		END_IF
	
		IF fb_ton_quitt.Q THEN
			fb_ton_quitt.IN := FALSE;
			fb_state_entry.i16_next_step := INIT;
		END_IF

END_CASE

fb_state_entry(i16_pos:= 2 );

fbGetUpsStatus(
	sNetId:= ,	(* wenn in AmsNetId nichts drin steht, wird immer die lokale genommen*)
	nPort:= 0,
	bEnable:= ,
	bValid=> , 
	bError=> , 
	nErrId=> ,
	stStatus=> );

IF st_config.b_config_fertig THEN
	(* Fehlermeldungen und Betriebsmeldungen ab dem Startindex in die globalen Meldungsarrays schreiben *)
	garr_stoermeldungen[st_config.i16_meld_startindex + 0] := FALSE;
	garr_stoermeldungen[st_config.i16_meld_startindex + 1] := FALSE;
	garr_stoermeldungen[st_config.i16_meld_startindex + 2] := FALSE;
	garr_stoermeldungen[st_config.i16_meld_startindex + 3] := FALSE;
	garr_stoermeldungen[st_config.i16_meld_startindex + 4] := FALSE;

	garr_betriebsmeldungen[st_config.i16_meld_startindex + 0] := bm_ReplaceBattery;
	garr_betriebsmeldungen[st_config.i16_meld_startindex + 1] := bm_NoPower;
	garr_betriebsmeldungen[st_config.i16_meld_startindex + 2] := bm_StatusNotValid;
	garr_betriebsmeldungen[st_config.i16_meld_startindex + 3] := FALSE;
	garr_betriebsmeldungen[st_config.i16_meld_startindex + 4] := FALSE;
END_IF
END_PROGRAM

(* POU EPT Lib/Programmbausteine/Routing/PC-Suche/ST_RoutingBackpanel, ST *)
PROGRAM ST_RoutingBackpanel
VAR_INPUT
	st_config						: struct_config;
	st_ctrl_in						: struct_ctrl_in;
END_VAR
VAR_OUTPUT
	st_ctrl_out					: struct_ctrl_out;
END_VAR
VAR
	fb_ton_wz					: TON;
	arr_read_routing_info			: ARRAY [0..31] OF ST_AmsRouteEntry;
	b_routing_station_gefunden		: BOOL;
	fb_add_route_entry			: FB_AddRouteEntry;
	fb_enum_route_entry			: FB_EnumRouteEntry;
	fb_ton_quitt					: TON;
	fb_state_entry					: ST_StateEntry;
	i16_eintrag					: INT := 0;
	b_ibn_start_routing			: BOOL := FALSE;
	fb_r_trig_ibn_start_routing		: R_TRIG;
	fb_ton_ibn_start_routing		: TON;
	s_backpanel_adresse			: STRING[255] := '';
	s_backpanel_netid			: STRING[255] := '';
	s_backpanel_name			: STRING[255] := '';
	s_temp_net_string				: STRING[255] := '';
	i16_temp_net_int				: INT := 0;
	s_temp_ip_string				: STRING[255] := '';
	i16_temp_ip_int				: INT := 0;
	s_temp_string_p11			: STRING[255] := '';
	s_temp_string_p12			: STRING[255] := '';
	s_temp_string_p13			: STRING[255] := '';
	fb_get_local_ams_netid		: ST_GetLocalAMSNetID;
	fb_get_adapters_info			: ST_GetAdaptersInfo;
	fb_get_host_name				: FB_GetHostName;
	fb_get_host_addr_by_name		: FB_GetHostAddrByName;
	st_pc_adapter_info			: ST_IpAdapterInfo;
	st_backpanel_adapter_info		: ST_IpAdapterInfo;
	sm_fehler_netid				: BOOL := FALSE;
	sm_fehler_adapter_info		: BOOL := FALSE;
	sm_fehler_host_name			: BOOL := FALSE;
	sm_fehler_host_addr			: BOOL := FALSE;
END_VAR
fb_ton_quitt(IN:= , PT:= t#100ms, Q=> , ET=> );
fb_ton_wz(IN:= , PT:= t#10s , Q=> , ET=> );

fb_r_trig_ibn_start_routing(CLK:= b_ibn_start_routing, Q=> );
fb_ton_ibn_start_routing(IN:= , PT:= t#1s, Q=> , ET=> );

IF fb_r_trig_ibn_start_routing.Q THEN
	fb_ton_ibn_start_routing.IN := TRUE;
ELSE
	IF fb_ton_ibn_start_routing.Q THEN
		b_ibn_start_routing := FALSE;
	 	fb_ton_ibn_start_routing.IN := FALSE;
	END_IF
END_IF

(* =======================================Toplevel========================================== *)
IF fb_state_entry.i16_next_step > INIT AND fb_state_entry.i16_next_step < FEHLER THEN
	 IF fb_get_adapters_info.bError OR fb_get_local_ams_netid.bError THEN
		fb_state_entry.i16_next_step := FEHLER;
	END_IF
END_IF

fb_state_entry(
	i16_next_step:= ,
	i16_pos:= 1,
	s_debugtext:= ,
	E=> ,
	X=> , 
	i16_step=> ,
	i16_last_step=> );

CASE fb_state_entry.i16_step OF
(*=======================================================*)
	0:
		fb_state_entry.i16_next_step := INIT;

(*=======================================================*)
	INIT:	(* Initialisierung *)
		st_ctrl_out.b_fehler := FALSE;
		st_ctrl_out.b_fertig := FALSE;
		st_ctrl_out.b_bereit := FALSE;
		fb_add_route_entry.bExecute := FALSE;
		fb_enum_route_entry.bExecute := FALSE;
		fb_enum_route_entry.eCmd := eEnumCmd_First;
		b_routing_station_gefunden := TRUE;
		i16_eintrag := 0;
		fb_get_local_ams_netid.bExecute := FALSE;
		fb_get_local_ams_netid.bQuit := FALSE;
		fb_get_adapters_info.bExecute := FALSE;
		fb_get_adapters_info.bQuit := FALSE;
		fb_get_host_name.bExecute := FALSE;
		fb_get_host_addr_by_name.bExecute := FALSE;
		sm_fehler_netid := FALSE;
		sm_fehler_adapter_info := FALSE;
		sm_fehler_host_name := FALSE;
		sm_fehler_host_addr := FALSE;

		FOR i16_eintrag := 0  TO (SIZEOF (arr_read_routing_info) / SIZEOF (arr_read_routing_info[0])) BY 1DO
			IF	i16_eintrag <32 THEN
				arr_read_routing_info[i16_eintrag].sName := '';
				arr_read_routing_info[i16_eintrag].sNetID := '';
				arr_read_routing_info[i16_eintrag].sAddress := '';
				arr_read_routing_info[i16_eintrag].eTransport := eRouteTransport_TCP_IP;
			END_IF
		END_FOR

		IF fb_get_local_ams_netid.bReady AND fb_get_adapters_info.bReady THEN
			fb_state_entry.i16_next_step := 20;
		END_IF

(*=======================================================*)
	20:	(* Die AMS-NetID des lokalen PC ermitteln *)
		IF fb_state_entry.E THEN
			fb_get_local_ams_netid.bExecute := TRUE;
		END_IF

		IF fb_get_local_ams_netid.bBusy THEN
			fb_get_local_ams_netid.bExecute := FALSE;
			fb_state_entry.i16_next_step := 20;
		END_IF

(*=======================================================*)
	30:
		IF NOT fb_get_local_ams_netid.bBusy  AND fb_get_local_ams_netid.bReady THEN
			IF NOT fb_get_local_ams_netid.bError THEN
				fb_state_entry.i16_next_step := 40;
			ELSE	(* Fehler *)
				sm_fehler_netid := TRUE;
				fb_state_entry.i16_next_step := 1000;
			END_IF
		END_IF

(*=======================================================*)
	40:	(* Ersten Routing Eintrag im Routingtable lesen *)
		IF fb_state_entry.E THEN
			s_temp_string_p11 := MID(fb_get_local_ams_netid.local_ams_netid, 1, 11);
			s_temp_string_p12 := MID(fb_get_local_ams_netid.local_ams_netid, 1, 12);
			s_temp_string_p13 := MID(fb_get_local_ams_netid.local_ams_netid, 1, 13);
			IF s_temp_string_p11 = '.' THEN
				(* Die vierte Zahl ist einstellig *)
				i16_temp_net_int := STRING_TO_INT(MID(fb_get_local_ams_netid.local_ams_netid, 1, 10));
			ELSIF s_temp_string_p12 = '.' THEN
				(* Die vierte Zahl ist zweistellig *)
				i16_temp_net_int := STRING_TO_INT(MID(fb_get_local_ams_netid.local_ams_netid, 2, 10));
			ELSIF s_temp_string_p13 = '.' THEN
				(* Die vierte Zahl ist dreistellig *)
				i16_temp_net_int := STRING_TO_INT(MID(fb_get_local_ams_netid.local_ams_netid, 3, 10));
			END_IF
			i16_temp_net_int := i16_temp_net_int  + 1;	(* Die NetID des Remote-Panel ist um 1 höher, als diejenige des PCs *)
			s_temp_net_string := INT_TO_STRING (i16_temp_net_int);
			s_backpanel_netid := CONCAT((CONCAT(MID(fb_get_local_ams_netid.s_ams_netid, 9, 1), s_temp_net_string)), '.1.1');
			fb_state_entry.i16_next_step := 50;
		END_IF

(*=======================================================*)
	50:	(* Die Adapter-Info des lokalen PC ermitteln *)
		IF fb_state_entry.E THEN
			fb_get_adapters_info.sNet_ID := fb_get_local_ams_netid.local_ams_netid;
			fb_get_adapters_info.bExecute := TRUE;
		END_IF

		IF fb_get_adapters_info.bBusy THEN
			fb_get_adapters_info.bExecute := FALSE;
			fb_state_entry.i16_next_step := 60;
		END_IF

(*=======================================================*)
	60:	(* Info steht zur Verfügung *)
		IF NOT fb_get_adapters_info.bBusy THEN
			IF NOT fb_get_adapters_info.bError THEN
				IF fb_get_adapters_info.bReady THEN
					st_pc_adapter_info := fb_get_adapters_info.st_ip_adapter_info;
					fb_state_entry.i16_next_step := 70;
				END_IF
			ELSE	(* Fehler *)
				sm_fehler_adapter_info := TRUE;
				fb_state_entry.i16_next_step := 1000;
			END_IF
		END_IF

(*=======================================================*)
	70:	(* Die Adapter-Info des Backpanel ermitteln *)
		IF fb_state_entry.E THEN
			fb_get_adapters_info.sNet_ID := s_backpanel_netid;
			fb_get_adapters_info.bExecute := TRUE;
		END_IF

		IF fb_get_adapters_info.bBusy THEN
			fb_get_adapters_info.bExecute := FALSE;
			fb_state_entry.i16_next_step := 80;
		END_IF

(*=======================================================*)
	80:	(* Info steht zur Verfügung *)
		IF NOT fb_get_adapters_info.bBusy THEN
			IF NOT fb_get_adapters_info.bError THEN
				IF fb_get_adapters_info.bReady THEN
					st_pc_adapter_info := fb_get_adapters_info.st_ip_adapter_info;
					s_backpanel_adresse := st_pc_adapter_info.sIpAddr;
					fb_state_entry.i16_next_step := 90;
				END_IF
			ELSE	(* Fehler *)
				sm_fehler_adapter_info := TRUE;
				fb_state_entry.i16_next_step := 1000;
			END_IF
		END_IF

(*=======================================================*)
	90:	(* Den Namen des Backpanels ermitteln *)
		IF fb_state_entry.E THEN
			fb_get_host_name.sNetID := s_backpanel_netid;
			fb_get_host_name.bExecute := TRUE;
		END_IF

		IF fb_get_host_name.bBusy THEN
			fb_get_host_name.bExecute := FALSE;
			fb_state_entry.i16_next_step := 100;
		END_IF

(*=======================================================*)
	100:	(* Info steht zur Verfügung *)
		IF NOT fb_get_host_name.bBusy THEN
			IF NOT fb_get_host_name.bError THEN
				s_backpanel_name := fb_get_host_name.sHostName;
				fb_state_entry.i16_next_step := 110;
			ELSE	(* Fehler *)
				sm_fehler_host_name := TRUE;
				fb_state_entry.i16_next_step := 1000;
			END_IF
		END_IF

(*=======================================================*)
	110:	(* Ersten Routing Eintrag im Routingtable lesen *)
		IF fb_state_entry.E THEN
			fb_enum_route_entry.bExecute := TRUE;
		END_IF

		IF fb_enum_route_entry.bBusy THEN
			fb_enum_route_entry.bExecute := FALSE;
			fb_state_entry.i16_next_step := 120;
		END_IF

(*=======================================================*)
	120:	(* Routinginformation ist vorhanden *)
		IF NOT fb_enum_route_entry.bBusy  THEN
			IF NOT fb_enum_route_entry.bError THEN
				IF NOT fb_enum_route_entry.bEOE THEN
					arr_read_routing_info[i16_eintrag] := fb_enum_route_entry.stRoute;
					fb_enum_route_entry.eCmd := eEnumCmd_Next;
					i16_eintrag := i16_eintrag + 1;
					fb_state_entry.i16_next_step := 110;
				ELSE	(* Alle vorhandenen Routingeinträge  wurden eingelesen*)
					fb_state_entry.i16_next_step := 130;
				END_IF
			ELSE	(* Fehler *)
				fb_state_entry.i16_next_step := 1000;
			END_IF
		END_IF

(*=======================================================*)
	130:	(* Alle Einträge sind gelesen *)
		IF fb_state_entry.E THEN
			(* Suche nach dem zugehörigen Backpanel *)
			FOR i16_eintrag := 0  TO (SIZEOF (arr_read_routing_info) / SIZEOF (arr_read_routing_info[0])) BY 1DO
				IF arr_read_routing_info[i16_eintrag].sNetID = s_backpanel_netid AND arr_read_routing_info[i16_eintrag].sAddress = s_backpanel_adresse THEN
					b_routing_station_gefunden := TRUE;
					fb_state_entry.i16_next_step :=  999;	(* Ende *)
					EXIT;
				ELSE
					b_routing_station_gefunden := FALSE;
				END_IF
			END_FOR
			IF NOT b_routing_station_gefunden THEN
				(* Station nicht in Liste -> eintragen *)
				fb_state_entry.i16_next_step := 140;
			END_IF
		END_IF

(*=======================================================*)
	140:	(* Routingtable mit Backpaneladresse füllen *)
		IF fb_state_entry.E THEN
			(* Initialisierung der Routingverbindung zum Backpanel *)
			fb_add_route_entry.stRoute.sName := s_backpanel_name;
			fb_add_route_entry.stRoute.sNetID := s_backpanel_netid;
			fb_add_route_entry.stRoute.sAddress := s_backpanel_adresse;
			fb_add_route_entry.stRoute.eTransport := eRouteTransport_TCP_IP;
			fb_add_route_entry.bExecute :=TRUE;
		END_IF

		IF fb_add_route_entry.bBusy THEN
			fb_add_route_entry.bExecute := FALSE;
			fb_state_entry.i16_next_step := 150;
		END_IF

(*=======================================================*)
	150:	(* Routingtable füllen läuft *)
		IF NOT fb_add_route_entry.bBusy THEN
			IF NOT fb_add_route_entry.bError THEN	(* Route wurde erfolgreich hinzugefügt *)
				fb_state_entry.i16_next_step := 999;
			ELSE	(* Fehler *)
				fb_state_entry.i16_next_step := 1000;
			END_IF
		END_IF

(*=======================================================*)
	999: (* Ende: Alle Stationen wurden im Routingtable eingetragen *)
		IF fb_r_trig_ibn_start_routing.Q THEN
			fb_state_entry.i16_next_step := INIT;
		END_IF

(*=======================================================*)
	1000: (* Fehler *)
		IF fb_state_entry.E THEN
			st_ctrl_out.b_fehler := TRUE;
			fb_ton_quitt.IN := FALSE;
			fb_add_route_entry.bExecute := FALSE;
			fb_enum_route_entry.bExecute := FALSE;
			fb_get_local_ams_netid.bExecute := FALSE;
			fb_get_local_ams_netid.bQuit := FALSE;
			fb_get_adapters_info.bExecute := FALSE;
			fb_get_adapters_info.bQuit := FALSE;
			fb_get_host_name.bExecute := FALSE;
			fb_get_host_addr_by_name.bExecute := FALSE;
		END_IF

		(*-----------------------Weiterschaltbedingungen----------------------------*)
		IF st_ctrl_in.b_quitt AND NOT fb_state_entry.E THEN
			st_ctrl_out.b_fehler := FALSE;
			fb_get_local_ams_netid .bQuit := TRUE;
			fb_get_adapters_info .bQuit := TRUE;
			fb_ton_quitt.IN := TRUE;
		END_IF

		IF fb_ton_quitt.Q OR  fb_r_trig_ibn_start_routing.Q THEN
			fb_ton_quitt.IN := FALSE;
			fb_state_entry.i16_next_step := INIT;
		END_IF
END_CASE

fb_state_entry(
	i16_next_step:= ,
	i16_pos:= 2,
	s_debugtext:= ,
	E=> ,
	X=> , 
	i16_step=> ,
	i16_last_step=> );

fb_get_local_ams_netid(
	bExecute:= , 
	bQuit:= , 
	bBusy=> , 
	bReady=> , 
	bError=> , 
	nErrId=> , 
	s_ams_netid=> );

fb_add_route_entry(
	sNetID:= '',
	stRoute:= ,
	bExecute:= ,
	tTimeout:= DEFAULT_ADS_TIMEOUT,
	bBusy=> ,
	bError=> ,
	nErrID=> );

fb_enum_route_entry(
	sNetID:= '',
	eCmd:= , 
	bExecute:= , 
	tTimeout:= DEFAULT_ADS_TIMEOUT,
	bBusy=> ,
	bError=> , 
	nErrID=> , 
	bEOE=> , 
	stRoute=> );

fb_get_adapters_info(
	sNet_ID:= , 
	bExecute:= , 
	bQuit:= , 
	bBusy=> ,
	bReady=> , 
	bError=> ,
	nErrId=> , 
	st_ip_adapter_info=> );

fb_get_host_name(
	sNetID:= ,
	bExecute:= , 
	tTimeout:= DEFAULT_ADS_TIMEOUT,
	bBusy=> , 
	bError=> ,
	nErrID=> , 
	sHostName=> );

fb_get_host_addr_by_name(
	sNetID:= '',
	sHostName:= ,
	bExecute:= , 
	tTimeout:= DEFAULT_ADS_TIMEOUT,
	bBusy=> , 
	bError=> , 
	nErrID=> , 
	sAddr=> , 
	arrAddr=> );

IF st_config.b_config_fertig THEN
	garr_stoermeldungen[st_config.i16_meld_startindex + 0] := sm_fehler_netid;
	garr_stoermeldungen[st_config.i16_meld_startindex + 1] := sm_fehler_adapter_info;
	garr_stoermeldungen[st_config.i16_meld_startindex + 2] := FALSE;
	garr_stoermeldungen[st_config.i16_meld_startindex + 3] := sm_fehler_host_addr;
	garr_stoermeldungen[st_config.i16_meld_startindex + 4] := FALSE;
	garr_stoermeldungen[st_config.i16_meld_startindex + 5] := FALSE;
	garr_stoermeldungen[st_config.i16_meld_startindex + 6] := FALSE;
	garr_stoermeldungen[st_config.i16_meld_startindex + 7] := FALSE;
	garr_stoermeldungen[st_config.i16_meld_startindex + 8] := FALSE;
	garr_stoermeldungen[st_config.i16_meld_startindex + 9] := FALSE;
	garr_stoermeldungen[st_config.i16_meld_startindex + 10] := FALSE;
	garr_stoermeldungen[st_config.i16_meld_startindex + 11] := FALSE;
	garr_stoermeldungen[st_config.i16_meld_startindex + 12] := FALSE;
	garr_stoermeldungen[st_config.i16_meld_startindex + 13] := FALSE;
	garr_stoermeldungen[st_config.i16_meld_startindex + 14] := FALSE;
	garr_stoermeldungen[st_config.i16_meld_startindex + 15] := FALSE;
	garr_stoermeldungen[st_config.i16_meld_startindex + 16] := FALSE;
	garr_stoermeldungen[st_config.i16_meld_startindex + 17] := FALSE;
	garr_stoermeldungen[st_config.i16_meld_startindex + 18] := FALSE;
	garr_stoermeldungen[st_config.i16_meld_startindex + 19] := FALSE;
	
	garr_betriebsmeldungen[st_config.i16_meld_startindex + 0] := FALSE;
	garr_betriebsmeldungen[st_config.i16_meld_startindex + 1] := FALSE;
	garr_betriebsmeldungen[st_config.i16_meld_startindex + 2] := FALSE;
	garr_betriebsmeldungen[st_config.i16_meld_startindex + 3] := FALSE;
	garr_betriebsmeldungen[st_config.i16_meld_startindex + 4] := FALSE;
	garr_betriebsmeldungen[st_config.i16_meld_startindex + 5] := FALSE;
	garr_betriebsmeldungen[st_config.i16_meld_startindex + 6] := FALSE;
	garr_betriebsmeldungen[st_config.i16_meld_startindex + 7] := FALSE;
	garr_betriebsmeldungen[st_config.i16_meld_startindex + 8] := FALSE;
	garr_betriebsmeldungen[st_config.i16_meld_startindex + 9] := FALSE;
	garr_betriebsmeldungen[st_config.i16_meld_startindex + 10] := FALSE;
	garr_betriebsmeldungen[st_config.i16_meld_startindex + 11] := FALSE;
	garr_betriebsmeldungen[st_config.i16_meld_startindex + 12] := FALSE;
	garr_betriebsmeldungen[st_config.i16_meld_startindex + 13] := FALSE;
	garr_betriebsmeldungen[st_config.i16_meld_startindex + 14] := FALSE;
	garr_betriebsmeldungen[st_config.i16_meld_startindex + 15] := FALSE;
	garr_betriebsmeldungen[st_config.i16_meld_startindex + 16] := FALSE;
	garr_betriebsmeldungen[st_config.i16_meld_startindex + 17] := FALSE;
	garr_betriebsmeldungen[st_config.i16_meld_startindex + 18] := FALSE;
	garr_betriebsmeldungen[st_config.i16_meld_startindex + 19] := FALSE;
END_IF
END_PROGRAM

(* POU EPT Lib/Programmbausteine/Routing/ST_GetAdaptersInfo, ST *)
FUNCTION_BLOCK ST_GetAdaptersInfo
VAR_INPUT
	sNet_ID						: T_AmsNetId;
	bExecute					: BOOL;
	bQuit						: BOOL;
END_VAR
VAR_OUTPUT
	bBusy						: BOOL;
	bReady						: BOOL;
	bError						: BOOL;
	nErrId						: UDINT;
	st_ip_adapter_info				: ST_IpAdapterInfo;
END_VAR
VAR
	fb_ton_quitt					: TON;
	fb_state_entry					: ST_StateEntry;
	fb_r_trig_execute				: R_TRIG;
	fb_get_adapters_info			: FB_GetAdaptersInfo;
	arr_adapters 					: ARRAY[0..MAX_LOCAL_ADAPTERS] OF ST_IpAdapterInfo;
END_VAR
(* Auslesen von IP-Adresse usw. des lokalen PCs *)
fb_r_trig_execute(CLK:= bExecute, Q=> );
fb_ton_quitt(IN:= , PT:= t#100ms, Q=> , ET=> );

(* =======================================Toplevel========================================== *)
IF fb_state_entry.i16_next_step > INIT AND fb_state_entry.i16_next_step < FEHLER THEN
	 IF fb_get_adapters_info.bError THEN
		fb_state_entry.i16_next_step := FEHLER;
	END_IF
END_IF

fb_state_entry(
	i16_next_step:= ,
	i16_pos:= 1,
	s_debugtext:= ,
	E=> ,
	X=> ,
	i16_step=> ,
	i16_last_step=> );

CASE fb_state_entry.i16_step OF
(*=======================================================*)
	0:
		fb_state_entry.i16_next_step := INIT;

(*=======================================================*)
	INIT:(* INIT *)
		bBusy := FALSE;
		bReady := FALSE;
		bError := FALSE;
		nErrId := 0;
		fb_get_adapters_info.bExecute := FALSE;
		fb_state_entry.i16_next_step := 20;

(*=======================================================*)
	20:	(* Warte auf Execute-Befehl *)
		IF fb_state_entry.E THEN
			bReady := TRUE;
		END_IF

		(*-----------------------Weiterschaltbedingungen----------------------------*)
		IF fb_r_trig_execute.Q THEN
			bReady := FALSE;
			bBusy := TRUE;
			fb_state_entry.i16_next_step := 30;
		END_IF

(*=======================================================*)
	30:	(* Starte mit Auslesen der Adapter-Info des lokalen PC *)
		IF fb_state_entry.E THEN
			fb_get_adapters_info.bExecute := TRUE;
		END_IF

		IF fb_get_adapters_info.bBusy THEN
			fb_get_adapters_info.bExecute := FALSE;
			fb_state_entry.i16_next_step := 40;
		END_IF

(*=======================================================*)
	40:	(* Adapter-Info wurde ausgelesen *)
		IF NOT fb_get_adapters_info.bBusy THEN
			IF NOT fb_get_adapters_info.bError THEN
				bBusy := FALSE;
				fb_state_entry.i16_next_step := 999;
			ELSE	(* Fehler *)
				fb_state_entry.i16_next_step := 1000;
			END_IF
		END_IF

(*=======================================================*)
	999:	(* Fertig *)
		st_ip_adapter_info := arr_adapters[1];
		fb_state_entry.i16_next_step := 20;

(*=======================================================*)
	FEHLER: (* Fehler *)
		IF fb_state_entry.E THEN
			bBusy := FALSE;
			bReady := FALSE;
			bError := TRUE;
			fb_get_adapters_info.bExecute := FALSE;
			fb_ton_quitt.IN := FALSE;
		END_IF

		(*-----------------------Weiterschaltbedingungen----------------------------*)
		IF bQuit AND NOT fb_state_entry.E THEN
			bError := FALSE;
			fb_ton_quitt.IN := TRUE;
			(* Quittierflanke für FB *)
			fb_get_adapters_info.bExecute := TRUE;
		END_IF

		IF fb_ton_quitt.Q THEN
			fb_ton_quitt.IN := FALSE;
			fb_state_entry.i16_next_step := INIT;
		END_IF
END_CASE

fb_state_entry(
	i16_next_step:= , 
	i16_pos:= 2,
	s_debugtext:= ,
	E=> ,
	X=> ,
	i16_step=> ,
	i16_last_step=> );

fb_get_adapters_info(
	sNetID:= sNet_ID,
	bExecute:= , 
	tTimeout:= DEFAULT_ADS_TIMEOUT,
	bBusy=> ,
	bError=> , 
	nErrID=> nErrId,
	arrAdapters=> arr_adapters,
	nCount=> , 
	nGet=> );
END_FUNCTION_BLOCK

(* POU Gemeinsamkeiten17xx/Programmbausteine/ST_Schreibe_Persistente_Daten, ST *)
PROGRAM ST_Schreibe_Persistente_Daten
VAR_INPUT
	bExecute			: BOOL;
	bQuit				: BOOL;
	t_schreibintervall		: TIME;
	b_steuerung_ein		: BOOL;
END_VAR
VAR_OUTPUT
	bBusy				: BOOL;
	bError				: BOOL;
	nErrId				: UDINT;
END_VAR
VAR
	fb_write_persistent_data		: FB_WritePersistentData;
	fb_ton_quitt					: TON;
	fb_state_entry				: ST_StateEntry;
	fb_ton_schreiben			: TON;
	fb_get_local_ams_netid		: ST_GetLocalAMSNetID;
	fb_r_trig_execute			: R_TRIG;
	fb_f_trig_steuerung			: F_TRIG;
	sm_fehler_daten_schreiben	: BOOL := FALSE;
	sm_fehler_netid				: BOOL := FALSE;

	gst_manuelles_bestueckprogramm_copy	: struct_bestueckprogramm;
	gst_PersDaten_Copy					: struct_PD;
END_VAR
(* Die Persistenten Daten der Maschine werden in einem wiederkehrenden Zeitintervall in eine Datei im TwinCAT Boot-Ordner geschrieben *)
fb_ton_quitt(IN:= , PT:= t#30s, Q=> , ET=> );
fb_ton_schreiben(IN:= , PT:= t_schreibintervall, Q=> , ET=> );

fb_r_trig_execute(CLK:= bExecute, Q=> );
fb_f_trig_steuerung(CLK:= b_steuerung_ein, Q=> );


fb_state_entry(	i16_pos:= 1 );

CASE fb_state_entry.i16_step OF
(*=======================================================*)
	INIT_OBJ:
		fb_state_entry.i16_next_step := INIT;

(*=======================================================*)
	INIT:
		IF fb_state_entry.E THEN
			bBusy := FALSE;
			bError := FALSE;
			fb_write_persistent_data.START := FALSE;
			fb_ton_schreiben.IN := FALSE;
			fb_get_local_ams_netid.bExecute := FALSE;
			fb_get_local_ams_netid .bQuit := FALSE;
			sm_fehler_daten_schreiben := FALSE;
			sm_fehler_netid := FALSE;
		END_IF

		fb_state_entry.i16_next_step := 20;

(*=======================================================*)
	20:	(* Die AMS-NetID des lokalen PC ermitteln *)
		IF fb_state_entry.E THEN
			fb_get_local_ams_netid.bExecute := TRUE;
		END_IF

		IF fb_get_local_ams_netid.bBusy THEN
			fb_get_local_ams_netid.bExecute := FALSE;
			fb_state_entry.i16_next_step := 30;
		END_IF

(*=======================================================*)
	30:
		IF NOT fb_get_local_ams_netid.bBusy  THEN
			IF NOT fb_get_local_ams_netid.bError THEN
				fb_state_entry.i16_next_step := BEREIT;
			ELSE	(* Fehler *)
				sm_fehler_netid := TRUE;
				fb_state_entry.i16_next_step := FEHLER;
			END_IF
		END_IF

(*=======================================================*)
	BEREIT:	(* Warte auf Freigabeflanke für zyklisches Schreiben der Daten /  Daten sichern, wenn Maschine ausgeschaltet wird *)
		IF 	fb_r_trig_execute.Q OR fb_f_trig_steuerung.Q THEN
			fb_state_entry.i16_next_step := 110;
		END_IF

		(*Schreibe bei einer Änderung*)
		IF	gi16_maschinenstatusinfo <> STATUS_MASCHINE_ARBEITET AND (
			(MEMCMP(ADR(gst_manuelles_bestueckprogramm_copy), ADR(gst_manuelles_bestueckprogramm), SIZEOF(gst_manuelles_bestueckprogramm_copy)) <> 0 ) OR
			(MEMCMP(ADR(gst_PersDaten_Copy), ADR(gst_PersDaten), SIZEOF(gst_PersDaten_Copy)) <> 0 ) 	) THEN
			gst_PersDaten_Copy:=gst_PersDaten;
			gst_manuelles_bestueckprogramm_copy:=gst_manuelles_bestueckprogramm;
			fb_state_entry.i16_next_step := 110;
		END_IF

(*=======================================================*)
	110:	(* Schreibe Persistente Daten *)
		IF fb_state_entry.E THEN
			bBusy := TRUE;
			fb_write_persistent_data.START := TRUE;
		END_IF

		IF fb_write_persistent_data.BUSY THEN
			fb_write_persistent_data.START := FALSE;
			fb_state_entry.i16_next_step := 120;
		END_IF

(*=======================================================*)
	120:	(* Daten wurden geschrieben *)
		IF NOT fb_write_persistent_data.BUSY  THEN
			IF NOT fb_write_persistent_data.ERR THEN
				bBusy := FALSE;
				fb_state_entry.i16_next_step := 100;
			ELSE
				sm_fehler_daten_schreiben := TRUE;
				fb_state_entry.i16_next_step := FEHLER;
			END_IF
		END_IF

(*=======================================================*)
	FEHLER:
		IF fb_state_entry.E THEN
			fb_ton_quitt.IN := TRUE;
			fb_get_local_ams_netid.bExecute := FALSE;
			fb_get_local_ams_netid.bQuit := FALSE;
			bError := TRUE;
		END_IF

		IF  fb_ton_quitt.Q THEN
			fb_ton_quitt.IN := FALSE;
			fb_get_local_ams_netid .bQuit := TRUE;
			fb_state_entry.i16_next_step := INIT;
		END_IF

END_CASE

fb_state_entry(i16_pos:= 2 );

fb_get_local_ams_netid(
	bExecute:= ,
	bQuit:= , 
	bBusy=> , 
	bReady=> , 
	bError=> , 
	nErrId=> , 
	s_ams_netid=> );

fb_write_persistent_data(
	NETID:= '',
	PORT:= 801,
	START:= , 
	TMOUT:= DEFAULT_ADS_TIMEOUT,
	MODE:= SPDM_2PASS,
	BUSY=> , 
	ERR=> , 
	ERRID=> );
END_PROGRAM

(* POU EPT Lib/Programmbausteine/ST_System_DateAndTime, ST *)
PROGRAM ST_System_DateAndTime
VAR
	w_year					: WORD := 16#0000;
	w_month					: WORD := 16#0000;
	w_day					: WORD := 16#0000;
	w_hour					: WORD := 16#0000;
	w_min					: WORD := 16#0000;
	w_sec					: WORD := 16#0000;
	fb_get_system_time 		: FB_LocalSystemTime;
END_VAR
(* =====Erzeugen der Systemzeit für die ganze Maschine======== *)
(* Die Umstellung von Sommer auf Winterzeit und umgekehrt erfolgt automatisch über die PC-Zeit *)
fb_get_system_time ( sNetID := '',
					bEnable 	:= TRUE,
					dwCycle 	:= 1,
					dwOpt	:= 1,
					tTimeout 	:= DEFAULT_ADS_TIMEOUT,
					bValid => b_system_time_valid,
					systemTime => gst_system_time, (* Systemzeit *)
					tzID 	=> );
(*=======================================================*)
gdt_system_time := SYSTEMTIME_TO_DT(fb_get_system_time.systemTime);

w_year:=gst_system_time.wYear;
w_month:=gst_system_time.wMonth;
w_day:=gst_system_time.wDay;
w_hour:=gst_system_time.wHour;
w_min:=gst_system_time.wMinute;
w_sec:=gst_system_time.wSecond;

gstr_system_time := '';
gstr_datum := '';
IF w_day < 10 THEN
	gstr_datum := CONCAT(gstr_datum ,WORD_TO_STRING(0));
END_IF;
gstr_datum := CONCAT(gstr_datum ,WORD_TO_STRING(w_day));
gstr_datum := CONCAT(gstr_datum , '.');

IF w_month < 10 THEN
	gstr_datum := CONCAT(gstr_datum ,WORD_TO_STRING(0));
END_IF;
gstr_datum := CONCAT(gstr_datum ,WORD_TO_STRING(w_month));
gstr_datum := CONCAT(gstr_datum , '.');
gstr_datum := CONCAT(gstr_datum ,WORD_TO_STRING(w_year));	(* Datum steht zur Verfügung *)

gstr_uhrzeit := '';
IF w_hour < 10 THEN
	gstr_uhrzeit := CONCAT(gstr_uhrzeit ,WORD_TO_STRING(0));
END_IF;
gstr_uhrzeit := CONCAT(gstr_uhrzeit ,WORD_TO_STRING(w_hour));
gstr_uhrzeit := CONCAT(gstr_uhrzeit , ':');

IF w_min < 10 THEN
	gstr_uhrzeit := CONCAT(gstr_uhrzeit ,WORD_TO_STRING(0));
END_IF;
gstr_uhrzeit := CONCAT(gstr_uhrzeit ,WORD_TO_STRING(w_min));
gstr_uhrzeit := CONCAT(gstr_uhrzeit , ':');

IF w_sec < 10 THEN
	gstr_uhrzeit := CONCAT(gstr_uhrzeit ,WORD_TO_STRING(0));
END_IF;
gstr_uhrzeit := CONCAT(gstr_uhrzeit ,WORD_TO_STRING(w_sec));	(* Uhrzeit steht zur Verfügung *)

gstr_system_time := CONCAT(gstr_system_time, gstr_datum );
gstr_system_time := CONCAT(gstr_system_time , ' ');
gstr_system_time := CONCAT(gstr_system_time , gstr_uhrzeit);	(* Ausgabe von Datum und Uhrzeit als String für z.B . die Visu *)
END_PROGRAM

(* POU Gemeinsamkeiten17xx/Allgemeines/ST_Tuerverriegelung, ST *)
PROGRAM ST_Tuerverriegelung
VAR_INPUT
	e_quittiertaste						: BOOL;
END_VAR
VAR
	fb_ton_wz						: TON;
	fb_r_trig_quitt						: R_TRIG;
	fb_f_trig_quitt						: F_TRIG;
	fb_blinker						: ST_Blinker;
	a_tuerverriegelung_vorne			AT %Q* : BOOL;
	a_tuerverriegelung_hinten			AT %Q* : BOOL;
	e_kontakt_tuerverriegelung_vorne	AT %I* : BOOL;
	e_kontakt_tuerverriegelung_hinten	AT %I* : BOOL;
END_VAR
(* Blinken *)
fb_blinker(
	b_start:= TRUE,
	t_taktzeit_on:=t#500ms,
	t_taktzeit_off:=t#500ms,
	b_blinker_out=> );

(* Zeiten *)
fb_ton_wz(IN:= , PT:= t#3s, Q=> , ET=> );

(* Flanken *)
fb_r_trig_quitt(CLK:= e_quittiertaste, Q=> );
fb_f_trig_quitt(CLK:= e_quittiertaste, Q=> );

(* Ansteuerung der Türverriegelung vorne und hinten *)
CASE gi16_betriebsart OF
	HAND:
		a_tuerverriegelung_vorne := FALSE;
		a_tuerverriegelung_hinten := FALSE;
	TIPPEN, AUTO:
		IF 	gi16_maschinenstatusinfo = STATUS_BETRIEBSBEREIT OR
			gi16_maschinenstatusinfo = STATUS_FEHLER
			THEN
				(* Türen freigeben *)
				a_tuerverriegelung_vorne := FALSE;
				a_tuerverriegelung_hinten := FALSE;
		ELSE
			(* Türen verriegelt, wenn geschlossen *)
			IF NOT e_kontakt_tuerverriegelung_vorne THEN
				a_tuerverriegelung_vorne := TRUE;
			END_IF
			IF NOT e_kontakt_tuerverriegelung_hinten THEN
				a_tuerverriegelung_hinten := TRUE;
			END_IF
		END_IF
END_CASE
END_PROGRAM

(* POU Gemeinsamkeiten17xx/Zylinder/ST_Zylinder, ST *)
PROGRAM ST_Zylinder
VAR
	b_first_cycle 			: BOOL := TRUE;
END_VAR
IF ST_BBGen.b_lesen_komplett THEN

	ST_Datainit_Zylinder();

	(* Zylinderaufrufe *)
	zyl_wt_zentrierer_tisch.fb(
		st_config:= ,
		bw_nocken_zylinder_einfahren:= ,
		bw_nocken_zylinder_ausfahren:= ,
		uw_nocken_zylinder_einfahren:= ,
		uw_nocken_zylinder_ausfahren:= ,
		b_direkttaste_ausfahren:= ,
		b_direkttaste_mittefahren:= ,
		b_direkttaste_einfahren	:= ,
		e_druckwaechter:= ST_Betriebsfreigaben.e_druckwaechter,
		i16_betriebsart:= gi16_betriebsart,
		b_no_gesteuert_im_norm_betrieb:= ,
		st_ctrl_in:= zyl_wt_zentrierer_tisch.st_ctrl.in,
		b_masterachse_hand_dialog_aktiv:= ,
		st_visu:= visu.st_zyl,
		st_ctrl_out=> zyl_wt_zentrierer_tisch.st_ctrl.out,
		a_ventil_einfahren=> ,
		a_ventil_ausfahren=> );
	
	zyl_wt_stopper_tisch.fb(
		st_config:= ,
		bw_nocken_zylinder_einfahren:= ,
		bw_nocken_zylinder_ausfahren:= ,
		uw_nocken_zylinder_einfahren:= ,
		uw_nocken_zylinder_ausfahren:= ,
		b_direkttaste_ausfahren:= ,
		b_direkttaste_mittefahren:= ,
		b_direkttaste_einfahren	:= ,
		e_druckwaechter:= ST_Betriebsfreigaben.e_druckwaechter,
		i16_betriebsart:= gi16_betriebsart,
		b_no_gesteuert_im_norm_betrieb:= ,
		st_ctrl_in:= zyl_wt_stopper_tisch.st_ctrl.in,
		b_masterachse_hand_dialog_aktiv:= ,
		st_visu:= visu.st_zyl,
		st_ctrl_out=> zyl_wt_stopper_tisch.st_ctrl.out,
		a_ventil_einfahren=> ,
		a_ventil_ausfahren=> );
	
	zyl_wt_stopper_auslauf.fb(
		st_config:= ,
		bw_nocken_zylinder_einfahren:= ,
		bw_nocken_zylinder_ausfahren:= ,
		uw_nocken_zylinder_einfahren:= ,
		uw_nocken_zylinder_ausfahren:= ,
		b_direkttaste_ausfahren:= ,
		b_direkttaste_mittefahren:= ,
		b_direkttaste_einfahren	:= ,
		e_druckwaechter:= ST_Betriebsfreigaben.e_druckwaechter,
		i16_betriebsart:= gi16_betriebsart,
		b_no_gesteuert_im_norm_betrieb:= ,
		st_ctrl_in:= zyl_wt_stopper_auslauf.st_ctrl.in,
		b_masterachse_hand_dialog_aktiv:= ,
		st_visu:= visu.st_zyl,
		st_ctrl_out=> zyl_wt_stopper_auslauf.st_ctrl.out,
		a_ventil_einfahren=> ,
		a_ventil_ausfahren=> );
	
	zyl_hublift_rechts_lift.fb(
		st_config:= ,
		bw_nocken_zylinder_einfahren:= ,
		bw_nocken_zylinder_ausfahren:= ,
		uw_nocken_zylinder_einfahren:= ,
		uw_nocken_zylinder_ausfahren:= ,
		b_direkttaste_ausfahren:= ,
		b_direkttaste_mittefahren:= ,
		b_direkttaste_einfahren	:= ,
		e_druckwaechter:= ST_Betriebsfreigaben.e_druckwaechter,
		i16_betriebsart:= gi16_betriebsart,
		b_no_gesteuert_im_norm_betrieb:= ,
		st_ctrl_in:= zyl_hublift_rechts_lift.st_ctrl.in,
		b_masterachse_hand_dialog_aktiv:= ,
		st_visu:= visu.st_zyl,
		st_ctrl_out=> zyl_hublift_rechts_lift.st_ctrl.out,
		a_ventil_einfahren=> ,
		a_ventil_ausfahren=> );
	
	zyl_hublift_rechts_wt_einzug.fb(
		st_config:= ,
		bw_nocken_zylinder_einfahren:= ,
		bw_nocken_zylinder_ausfahren:= ,
		uw_nocken_zylinder_einfahren:= ,
		uw_nocken_zylinder_ausfahren:= ,
		b_direkttaste_ausfahren:= ,
		b_direkttaste_mittefahren:= ,
		b_direkttaste_einfahren	:= ,
		e_druckwaechter:= ST_Betriebsfreigaben.e_druckwaechter,
		i16_betriebsart:= gi16_betriebsart,
		b_no_gesteuert_im_norm_betrieb:= ,
		st_ctrl_in:= zyl_hublift_rechts_wt_einzug.st_ctrl.in,
		b_masterachse_hand_dialog_aktiv:= ,
		st_visu:= visu.st_zyl,
		st_ctrl_out=> zyl_hublift_rechts_wt_einzug.st_ctrl.out,
		a_ventil_einfahren=> ,
		a_ventil_ausfahren=> );
	
	zyl_hublift_rechts_wt_klinke.fb(
		st_config:= ,
		bw_nocken_zylinder_einfahren:= ,
		bw_nocken_zylinder_ausfahren:= ,
		uw_nocken_zylinder_einfahren:= ,
		uw_nocken_zylinder_ausfahren:= ,
		b_direkttaste_ausfahren:= ,
		b_direkttaste_mittefahren:= ,
		b_direkttaste_einfahren	:= ,
		e_druckwaechter:= ST_Betriebsfreigaben.e_druckwaechter,
		i16_betriebsart:= gi16_betriebsart,
		b_no_gesteuert_im_norm_betrieb:= ,
		st_ctrl_in:= zyl_hublift_rechts_wt_klinke.st_ctrl.in,
		b_masterachse_hand_dialog_aktiv:= ,
		st_visu:= visu.st_zyl,
		st_ctrl_out=> zyl_hublift_rechts_wt_klinke.st_ctrl.out,
		a_ventil_einfahren=> ,
		a_ventil_ausfahren=> );
	
	zyl_hublift_links_lift.fb(
		st_config:= ,
		bw_nocken_zylinder_einfahren:= ,
		bw_nocken_zylinder_ausfahren:= ,
		uw_nocken_zylinder_einfahren:= ,
		uw_nocken_zylinder_ausfahren:= ,
		b_direkttaste_ausfahren:= ,
		b_direkttaste_mittefahren:= ,
		b_direkttaste_einfahren	:= ,
		e_druckwaechter:= ST_Betriebsfreigaben.e_druckwaechter,
		i16_betriebsart:= gi16_betriebsart,
		b_no_gesteuert_im_norm_betrieb:= ,
		st_ctrl_in:= zyl_hublift_links_lift.st_ctrl.in,
		b_masterachse_hand_dialog_aktiv:= ,
		st_visu:= visu.st_zyl,
		st_ctrl_out=> zyl_hublift_links_lift.st_ctrl.out,
		a_ventil_einfahren=> ,
		a_ventil_ausfahren=> );
	
	zyl_hublift_links_wt_einzug.fb(
		st_config:= ,
		bw_nocken_zylinder_einfahren:= ,
		bw_nocken_zylinder_ausfahren:= ,
		uw_nocken_zylinder_einfahren:= ,
		uw_nocken_zylinder_ausfahren:= ,
		b_direkttaste_ausfahren:= ,
		b_direkttaste_mittefahren:= ,
		b_direkttaste_einfahren	:= ,
		e_druckwaechter:= ST_Betriebsfreigaben.e_druckwaechter,
		i16_betriebsart:= gi16_betriebsart,
		b_no_gesteuert_im_norm_betrieb:= ,
		st_ctrl_in:= zyl_hublift_links_wt_einzug.st_ctrl.in,
		b_masterachse_hand_dialog_aktiv:= ,
		st_visu:= visu.st_zyl,
		st_ctrl_out=> zyl_hublift_links_wt_einzug.st_ctrl.out,
		a_ventil_einfahren=> ,
		a_ventil_ausfahren=> );
	
	zyl_hublift_links_wt_klinke.fb(
		st_config:= ,
		bw_nocken_zylinder_einfahren:= ,
		bw_nocken_zylinder_ausfahren:= ,
		uw_nocken_zylinder_einfahren:= ,
		uw_nocken_zylinder_ausfahren:= ,
		b_direkttaste_ausfahren:= ,
		b_direkttaste_mittefahren:= ,
		b_direkttaste_einfahren	:= ,
		e_druckwaechter:= ST_Betriebsfreigaben.e_druckwaechter,
		i16_betriebsart:= gi16_betriebsart,
		b_no_gesteuert_im_norm_betrieb:= ,
		st_ctrl_in:= zyl_hublift_links_wt_klinke.st_ctrl.in,
		b_masterachse_hand_dialog_aktiv:= ,
		st_visu:= visu.st_zyl,
		st_ctrl_out=> zyl_hublift_links_wt_klinke.st_ctrl.out,
		a_ventil_einfahren=> ,
		a_ventil_ausfahren=> );
	
	zyl_hublift_links_stopper.fb(
		st_config:= ,
		bw_nocken_zylinder_einfahren:= ,
		bw_nocken_zylinder_ausfahren:= ,
		uw_nocken_zylinder_einfahren:= ,
		uw_nocken_zylinder_ausfahren:= ,
		b_direkttaste_ausfahren:= ,
		b_direkttaste_mittefahren:= ,
		b_direkttaste_einfahren	:= ,
		e_druckwaechter:= ST_Betriebsfreigaben.e_druckwaechter,
		i16_betriebsart:= gi16_betriebsart,
		b_no_gesteuert_im_norm_betrieb:= ,
		st_ctrl_in:= zyl_hublift_links_stopper.st_ctrl.in,
		b_masterachse_hand_dialog_aktiv:= ,
		st_visu:= visu.st_zyl,
		st_ctrl_out=> zyl_hublift_links_stopper.st_ctrl.out,
		a_ventil_einfahren=> ,
		a_ventil_ausfahren=> );
	
	zyl_hublift_links_eingriffschutz.fb(
		st_config:= ,
		bw_nocken_zylinder_einfahren:= ,
		bw_nocken_zylinder_ausfahren:= ,
		uw_nocken_zylinder_einfahren:= ,
		uw_nocken_zylinder_ausfahren:= ,
		b_direkttaste_ausfahren:= ,
		b_direkttaste_mittefahren:= ,
		b_direkttaste_einfahren	:= ,
		e_druckwaechter:= ST_Betriebsfreigaben.e_druckwaechter,
		i16_betriebsart:= gi16_betriebsart,
		b_no_gesteuert_im_norm_betrieb:= ,
		st_ctrl_in:= zyl_hublift_links_eingriffschutz.st_ctrl.in,
		b_masterachse_hand_dialog_aktiv:= ,
		st_visu:= visu.st_zyl,
		st_ctrl_out=> zyl_hublift_links_eingriffschutz.st_ctrl.out,
		a_ventil_einfahren=> ,
		a_ventil_ausfahren=> );
	
	CASE gst_datensatz.st_md.i16_typ_zelle OF
		KEINE_ZELLE:
			;
	
		BESTUECKZELLE_1700:
			zyl_bawe_faenger_li.fb.st_config.b_aktiv := NOT gst_datensatz.st_md.b_wt_transport_simulation;
			zyl_bawe_faenger_li.fb(
				st_config:= ,
				bw_nocken_zylinder_einfahren:= ,
				bw_nocken_zylinder_ausfahren:= ,
				uw_nocken_zylinder_einfahren:= ,
				uw_nocken_zylinder_ausfahren:= ,
				b_direkttaste_ausfahren:= ,
				b_direkttaste_mittefahren:= ,
				b_direkttaste_einfahren	:= ,
				e_druckwaechter:= ST_Betriebsfreigaben.e_druckwaechter,
				i16_betriebsart:= gi16_betriebsart,
				b_no_gesteuert_im_norm_betrieb:= ,
				st_ctrl_in:= zyl_bawe_faenger_li.st_ctrl.in,
				b_masterachse_hand_dialog_aktiv:= ,
				st_visu:= visu.st_zyl,
				st_ctrl_out=> zyl_bawe_faenger_li.st_ctrl.out,
				a_ventil_einfahren=> ,
				a_ventil_ausfahren=> );
	
			zyl_bawe_faenger_re.fb.st_config.b_aktiv := NOT gst_datensatz.st_md.b_wt_transport_simulation;
			zyl_bawe_faenger_re.fb(
				st_config:= ,
				bw_nocken_zylinder_einfahren:= ,
				bw_nocken_zylinder_ausfahren:= ,
				uw_nocken_zylinder_einfahren:= ,
				uw_nocken_zylinder_ausfahren:= ,
				b_direkttaste_ausfahren:= ,
				b_direkttaste_mittefahren:= ,
				b_direkttaste_einfahren	:= ,
				e_druckwaechter:= ST_Betriebsfreigaben.e_druckwaechter,
				i16_betriebsart:= gi16_betriebsart,
				b_no_gesteuert_im_norm_betrieb:= ,
				st_ctrl_in:= zyl_bawe_faenger_re.st_ctrl.in,
				b_masterachse_hand_dialog_aktiv:= ,
				st_visu:= visu.st_zyl,
				st_ctrl_out=> zyl_bawe_faenger_re.st_ctrl.out,
				a_ventil_einfahren=> ,
				a_ventil_ausfahren=> );
	
			zyl_bawe_halter_li.fb.st_config.b_aktiv := NOT gst_datensatz.st_md.b_wt_transport_simulation;
			zyl_bawe_halter_li.fb(
				st_config:= ,
				bw_nocken_zylinder_einfahren:= ,
				bw_nocken_zylinder_ausfahren:= ,
				uw_nocken_zylinder_einfahren:= ,
				uw_nocken_zylinder_ausfahren:= ,
				b_direkttaste_ausfahren:= ,
				b_direkttaste_mittefahren:= ,
				b_direkttaste_einfahren	:= ,
				e_druckwaechter:= ST_Betriebsfreigaben.e_druckwaechter,
				i16_betriebsart:= gi16_betriebsart,
				b_no_gesteuert_im_norm_betrieb:= ,
				st_ctrl_in:= zyl_bawe_halter_li.st_ctrl.in,
				b_masterachse_hand_dialog_aktiv:= ,
				st_visu:= visu.st_zyl,
				st_ctrl_out=> zyl_bawe_halter_li.st_ctrl.out,
				a_ventil_einfahren=> ,
				a_ventil_ausfahren=> );
	
			zyl_bawe_halter_re.fb.st_config.b_aktiv := NOT gst_datensatz.st_md.b_wt_transport_simulation;
			zyl_bawe_halter_re.fb(
				st_config:= ,
				bw_nocken_zylinder_einfahren:= ,
				bw_nocken_zylinder_ausfahren:= ,
				uw_nocken_zylinder_einfahren:= ,
				uw_nocken_zylinder_ausfahren:= ,
				b_direkttaste_ausfahren:= ,
				b_direkttaste_mittefahren:= ,
				b_direkttaste_einfahren	:= ,
				e_druckwaechter:= ST_Betriebsfreigaben.e_druckwaechter,
				i16_betriebsart:= gi16_betriebsart,
				b_no_gesteuert_im_norm_betrieb:= ,
				st_ctrl_in:= zyl_bawe_halter_re.st_ctrl.in,
				b_masterachse_hand_dialog_aktiv:= ,
				st_visu:= visu.st_zyl,
				st_ctrl_out=> zyl_bawe_halter_re.st_ctrl.out,
				a_ventil_einfahren=> ,
				a_ventil_ausfahren=> );
	
			zyl_bawe_querschub.fb.st_config.b_aktiv := NOT gst_datensatz.st_md.b_wt_transport_simulation;
			zyl_bawe_querschub.fb(
				st_config:= ,
				bw_nocken_zylinder_einfahren:= ,
				bw_nocken_zylinder_ausfahren:= ,
				uw_nocken_zylinder_einfahren:= ,
				uw_nocken_zylinder_ausfahren:= ,
				b_direkttaste_ausfahren:= ,
				b_direkttaste_mittefahren:= ,
				b_direkttaste_einfahren	:= ,
				e_druckwaechter:= ST_Betriebsfreigaben.e_druckwaechter,
				i16_betriebsart:= gi16_betriebsart,
				b_no_gesteuert_im_norm_betrieb:= ,
				st_ctrl_in:= zyl_bawe_querschub.st_ctrl.in,
				b_masterachse_hand_dialog_aktiv:= ,
				st_visu:= visu.st_zyl,
				st_ctrl_out=> zyl_bawe_querschub.st_ctrl.out,
				a_ventil_einfahren=> ,
				a_ventil_ausfahren=> );
	
			zyl_bawe_vorschub.fb.st_config.b_aktiv := NOT gst_datensatz.st_md.b_wt_transport_simulation;
			zyl_bawe_vorschub.fb(
				st_config:= ,
				bw_nocken_zylinder_einfahren:= ,
				bw_nocken_zylinder_ausfahren:= ,
				uw_nocken_zylinder_einfahren:= ,
				uw_nocken_zylinder_ausfahren:= ,
				b_direkttaste_ausfahren:= ,
				b_direkttaste_mittefahren:= ,
				b_direkttaste_einfahren	:= ,
				e_druckwaechter:= ST_Betriebsfreigaben.e_druckwaechter,
				i16_betriebsart:= gi16_betriebsart,
				b_no_gesteuert_im_norm_betrieb:= ,
				st_ctrl_in:= zyl_bawe_vorschub.st_ctrl.in,
				b_masterachse_hand_dialog_aktiv:= ,
				st_visu:= visu.st_zyl,
				st_ctrl_out=> zyl_bawe_vorschub.st_ctrl.out,
				a_ventil_einfahren=> a_zyl_vorschub_einfahren,
				a_ventil_ausfahren=> a_zyl_vorschub_ausfahren);
			
			zyl_haspel_li_heben.fb(
				st_config:= ,
				bw_nocken_zylinder_einfahren:= ,
				bw_nocken_zylinder_ausfahren:= ,
				uw_nocken_zylinder_einfahren:= ,
				uw_nocken_zylinder_ausfahren:= ,
				b_direkttaste_ausfahren:= ,
				b_direkttaste_mittefahren:= ,
				b_direkttaste_einfahren	:= ,
				e_druckwaechter:= ST_Betriebsfreigaben.e_druckwaechter,
				i16_betriebsart:= gi16_betriebsart,
				b_no_gesteuert_im_norm_betrieb:= ,
				st_ctrl_in:= zyl_haspel_li_heben.st_ctrl.in,
				b_masterachse_hand_dialog_aktiv:= ,
				st_visu:= visu.st_zyl,
				st_ctrl_out=> zyl_haspel_li_heben.st_ctrl.out,
				a_ventil_einfahren=> ,
				a_ventil_ausfahren=> );
	
			zyl_haspel_li_abspulen.fb(
				st_config:= ,
				bw_nocken_zylinder_einfahren:= ,
				bw_nocken_zylinder_ausfahren:= ,
				uw_nocken_zylinder_einfahren:= ,
				uw_nocken_zylinder_ausfahren:= ,
				b_direkttaste_ausfahren:= ,
				b_direkttaste_mittefahren:= ,
				b_direkttaste_einfahren	:= ,
				e_druckwaechter:= ST_Betriebsfreigaben.e_druckwaechter,
				i16_betriebsart:= gi16_betriebsart,
				b_no_gesteuert_im_norm_betrieb:= ,
				st_ctrl_in:= zyl_haspel_li_abspulen.st_ctrl.in,
				b_masterachse_hand_dialog_aktiv:= ,
				st_visu:= visu.st_zyl,
				st_ctrl_out=> zyl_haspel_li_abspulen.st_ctrl.out,
				a_ventil_einfahren=> ,
				a_ventil_ausfahren=> );
			
			zyl_haspel_li_sperren.fb(
				st_config:= ,
				bw_nocken_zylinder_einfahren:= ,
				bw_nocken_zylinder_ausfahren:= ,
				uw_nocken_zylinder_einfahren:= ,
				uw_nocken_zylinder_ausfahren:= ,
				b_direkttaste_ausfahren:= ,
				b_direkttaste_mittefahren:= ,
				b_direkttaste_einfahren	:= ,
				e_druckwaechter:= ST_Betriebsfreigaben.e_druckwaechter,
				i16_betriebsart:= gi16_betriebsart,
				b_no_gesteuert_im_norm_betrieb:= ,
				st_ctrl_in:= zyl_haspel_li_sperren.st_ctrl.in,
				b_masterachse_hand_dialog_aktiv:= ,
				st_visu:= visu.st_zyl,
				st_ctrl_out=> zyl_haspel_li_sperren.st_ctrl.out,
				a_ventil_einfahren=> ,
				a_ventil_ausfahren=> );
			
			zyl_haspel_re_heben.fb(
				st_config:= ,
				bw_nocken_zylinder_einfahren:= ,
				bw_nocken_zylinder_ausfahren:= ,
				uw_nocken_zylinder_einfahren:= ,
				uw_nocken_zylinder_ausfahren:= ,
				b_direkttaste_ausfahren:= ,
				b_direkttaste_mittefahren:= ,
				b_direkttaste_einfahren	:= ,
				e_druckwaechter:= ST_Betriebsfreigaben.e_druckwaechter,
				i16_betriebsart:= gi16_betriebsart,
				b_no_gesteuert_im_norm_betrieb:= ,
				st_ctrl_in:= zyl_haspel_re_heben.st_ctrl.in,
				b_masterachse_hand_dialog_aktiv:= ,
				st_visu:= visu.st_zyl,
				st_ctrl_out=> zyl_haspel_re_heben.st_ctrl.out,
				a_ventil_einfahren=> ,
				a_ventil_ausfahren=> );
			
			zyl_haspel_re_abspulen.fb(
				st_config:= ,
				bw_nocken_zylinder_einfahren:= ,
				bw_nocken_zylinder_ausfahren:= ,
				uw_nocken_zylinder_einfahren:= ,
				uw_nocken_zylinder_ausfahren:= ,
				b_direkttaste_ausfahren:= ,
				b_direkttaste_mittefahren:= ,
				b_direkttaste_einfahren	:= ,
				e_druckwaechter:= ST_Betriebsfreigaben.e_druckwaechter,
				i16_betriebsart:= gi16_betriebsart,
				b_no_gesteuert_im_norm_betrieb:= ,
				st_ctrl_in:= zyl_haspel_re_abspulen.st_ctrl.in,
				b_masterachse_hand_dialog_aktiv:= ,
				st_visu:= visu.st_zyl,
				st_ctrl_out=> zyl_haspel_re_abspulen.st_ctrl.out,
				a_ventil_einfahren=> ,
				a_ventil_ausfahren=> );
			
			zyl_haspel_re_sperren.fb(
				st_config:= ,
				bw_nocken_zylinder_einfahren:= ,
				bw_nocken_zylinder_ausfahren:= ,
				uw_nocken_zylinder_einfahren:= ,
				uw_nocken_zylinder_ausfahren:= ,
				b_direkttaste_ausfahren:= ,
				b_direkttaste_mittefahren:= ,
				b_direkttaste_einfahren	:= ,
				e_druckwaechter:= ST_Betriebsfreigaben.e_druckwaechter,
				i16_betriebsart:= gi16_betriebsart,
				b_no_gesteuert_im_norm_betrieb:= ,
				st_ctrl_in:= zyl_haspel_re_sperren.st_ctrl.in,
				b_masterachse_hand_dialog_aktiv:= ,
				st_visu:= visu.st_zyl,
				st_ctrl_out=> zyl_haspel_re_sperren.st_ctrl.out,
				a_ventil_einfahren=> ,
				a_ventil_ausfahren=> );
			
			zyl_haspel_verschieben.fb(
				st_config:= ,
				bw_nocken_zylinder_einfahren:= ,
				bw_nocken_zylinder_ausfahren:= ,
				uw_nocken_zylinder_einfahren:= ,
				uw_nocken_zylinder_ausfahren:= ,
				b_direkttaste_ausfahren:= ,
				b_direkttaste_mittefahren:= ,
				b_direkttaste_einfahren	:= ,
				e_druckwaechter:= ST_Betriebsfreigaben.e_druckwaechter,
				i16_betriebsart:= gi16_betriebsart,
				b_no_gesteuert_im_norm_betrieb:= ,
				st_ctrl_in:= zyl_haspel_verschieben.st_ctrl.in,
				b_masterachse_hand_dialog_aktiv:= ,
				st_visu:= visu.st_zyl,
				st_ctrl_out=> zyl_haspel_verschieben.st_ctrl.out,
				a_ventil_einfahren=> ,
				a_ventil_ausfahren=> );

			zyl_bandeinzuege_verschieben.fb(
				st_config:= ,
				bw_nocken_zylinder_einfahren:= ,
				bw_nocken_zylinder_ausfahren:= ,
				uw_nocken_zylinder_einfahren:= ,
				uw_nocken_zylinder_ausfahren:= ,
				b_direkttaste_ausfahren:= ,
				b_direkttaste_mittefahren:= ,
				b_direkttaste_einfahren	:= ,
				e_druckwaechter:= ST_Betriebsfreigaben.e_druckwaechter,
				i16_betriebsart:= gi16_betriebsart,
				b_no_gesteuert_im_norm_betrieb:= ,
				st_ctrl_in:= zyl_bandeinzuege_verschieben.st_ctrl.in,
				b_masterachse_hand_dialog_aktiv:= ,
				st_visu:= visu.st_zyl,
				st_ctrl_out=> zyl_bandeinzuege_verschieben.st_ctrl.out,
				a_ventil_einfahren=> ,
				a_ventil_ausfahren=> );
	

		(*	zyl_Indexier_Bestueckpos.fb.st_config.b_aktiv := NOT gst_datensatz.st_md.b_wt_transport_simulation;*)
			zyl_Indexier_Bestueckpos.fb(
				st_config:= ,
				bw_nocken_zylinder_einfahren:= ,
				bw_nocken_zylinder_ausfahren:= ,
				uw_nocken_zylinder_einfahren:= ,
				uw_nocken_zylinder_ausfahren:= ,
				b_direkttaste_ausfahren:= ,
				b_direkttaste_mittefahren:= ,
				b_direkttaste_einfahren	:= ,
				e_druckwaechter:= ST_Betriebsfreigaben.e_druckwaechter,
				i16_betriebsart:= gi16_betriebsart,
				b_no_gesteuert_im_norm_betrieb:= ,
				st_ctrl_in:= zyl_Indexier_Bestueckpos.st_ctrl.in,
				b_masterachse_hand_dialog_aktiv:= ,
				st_visu:= visu.st_zyl,
				st_ctrl_out=> zyl_Indexier_Bestueckpos.st_ctrl.out,
				a_ventil_einfahren=> ,
				a_ventil_ausfahren=> );
	
		(*	zyl_Indexier_Einlauf.fb.st_config.b_aktiv := NOT gst_datensatz.st_md.b_wt_transport_simulation;*)
			zyl_Indexier_Einlauf.fb(
				st_config:= ,
				bw_nocken_zylinder_einfahren:= ,
				bw_nocken_zylinder_ausfahren:= ,
				uw_nocken_zylinder_einfahren:= ,
				uw_nocken_zylinder_ausfahren:= ,
				b_direkttaste_ausfahren:= ,
				b_direkttaste_mittefahren:= ,
				b_direkttaste_einfahren	:= ,
				e_druckwaechter:= ST_Betriebsfreigaben.e_druckwaechter,
				i16_betriebsart:= gi16_betriebsart,
				b_no_gesteuert_im_norm_betrieb:= ,
				st_ctrl_in:= zyl_Indexier_Einlauf.st_ctrl.in,
				b_masterachse_hand_dialog_aktiv:= ,
				st_visu:= visu.st_zyl,
				st_ctrl_out=> zyl_Indexier_Einlauf.st_ctrl.out,
				a_ventil_einfahren=> ,
				a_ventil_ausfahren=> );

		BESTUECKZELLE_1720:
			zyl_wt_stopper_einlauf.fb(
				st_config:= ,
				bw_nocken_zylinder_einfahren:= ,
				bw_nocken_zylinder_ausfahren:= ,
				uw_nocken_zylinder_einfahren:= ,
				uw_nocken_zylinder_ausfahren:= ,
				b_direkttaste_ausfahren:= ,
				b_direkttaste_mittefahren:= ,
				b_direkttaste_einfahren	:= ,
				e_druckwaechter:= ST_Betriebsfreigaben.e_druckwaechter,
				i16_betriebsart:= gi16_betriebsart,
				b_no_gesteuert_im_norm_betrieb:= ,
				st_ctrl_in:= zyl_wt_stopper_einlauf.st_ctrl.in,
				b_masterachse_hand_dialog_aktiv:= ,
				st_visu:= visu.st_zyl,
				st_ctrl_out=> zyl_wt_stopper_einlauf.st_ctrl.out,
				a_ventil_einfahren=> ,
				a_ventil_ausfahren=> );
	
			zyl_haspel_li_heben.fb(
				st_config:= ,
				bw_nocken_zylinder_einfahren:= ,
				bw_nocken_zylinder_ausfahren:= ,
				uw_nocken_zylinder_einfahren:= ,
				uw_nocken_zylinder_ausfahren:= ,
				b_direkttaste_ausfahren:= ,
				b_direkttaste_mittefahren:= ,
				b_direkttaste_einfahren	:= ,
				e_druckwaechter:= ST_Betriebsfreigaben.e_druckwaechter,
				i16_betriebsart:= gi16_betriebsart,
				b_no_gesteuert_im_norm_betrieb:= ,
				st_ctrl_in:= zyl_haspel_li_heben.st_ctrl.in,
				b_masterachse_hand_dialog_aktiv:= ,
				st_visu:= visu.st_zyl,
				st_ctrl_out=> zyl_haspel_li_heben.st_ctrl.out,
				a_ventil_einfahren=> ,
				a_ventil_ausfahren=> );
			
			zyl_haspel_li_abspulen.fb(
				st_config:= ,
				bw_nocken_zylinder_einfahren:= ,
				bw_nocken_zylinder_ausfahren:= ,
				uw_nocken_zylinder_einfahren:= ,
				uw_nocken_zylinder_ausfahren:= ,
				b_direkttaste_ausfahren:= ,
				b_direkttaste_mittefahren:= ,
				b_direkttaste_einfahren	:= ,
				e_druckwaechter:= ST_Betriebsfreigaben.e_druckwaechter,
				i16_betriebsart:= gi16_betriebsart,
				b_no_gesteuert_im_norm_betrieb:= ,
				st_ctrl_in:= zyl_haspel_li_abspulen.st_ctrl.in,
				b_masterachse_hand_dialog_aktiv:= ,
				st_visu:= visu.st_zyl,
				st_ctrl_out=> zyl_haspel_li_abspulen.st_ctrl.out,
				a_ventil_einfahren=> ,
				a_ventil_ausfahren=> );
			
			zyl_haspel_li_sperren.fb(
				st_config:= ,
				bw_nocken_zylinder_einfahren:= ,
				bw_nocken_zylinder_ausfahren:= ,
				uw_nocken_zylinder_einfahren:= ,
				uw_nocken_zylinder_ausfahren:= ,
				b_direkttaste_ausfahren:= ,
				b_direkttaste_mittefahren:= ,
				b_direkttaste_einfahren	:= ,
				e_druckwaechter:= ST_Betriebsfreigaben.e_druckwaechter,
				i16_betriebsart:= gi16_betriebsart,
				b_no_gesteuert_im_norm_betrieb:= ,
				st_ctrl_in:= zyl_haspel_li_sperren.st_ctrl.in,
				b_masterachse_hand_dialog_aktiv:= ,
				st_visu:= visu.st_zyl,
				st_ctrl_out=> zyl_haspel_li_sperren.st_ctrl.out,
				a_ventil_einfahren=> ,
				a_ventil_ausfahren=> );
			
			zyl_haspel_re_heben.fb(
				st_config:= ,
				bw_nocken_zylinder_einfahren:= ,
				bw_nocken_zylinder_ausfahren:= ,
				uw_nocken_zylinder_einfahren:= ,
				uw_nocken_zylinder_ausfahren:= ,
				b_direkttaste_ausfahren:= ,
				b_direkttaste_mittefahren:= ,
				b_direkttaste_einfahren	:= ,
				e_druckwaechter:= ST_Betriebsfreigaben.e_druckwaechter,
				i16_betriebsart:= gi16_betriebsart,
				b_no_gesteuert_im_norm_betrieb:= ,
				st_ctrl_in:= zyl_haspel_re_heben.st_ctrl.in,
				b_masterachse_hand_dialog_aktiv:= ,
				st_visu:= visu.st_zyl,
				st_ctrl_out=> zyl_haspel_re_heben.st_ctrl.out,
				a_ventil_einfahren=> ,
				a_ventil_ausfahren=> );
			
			zyl_haspel_re_abspulen.fb(
				st_config:= ,
				bw_nocken_zylinder_einfahren:= ,
				bw_nocken_zylinder_ausfahren:= ,
				uw_nocken_zylinder_einfahren:= ,
				uw_nocken_zylinder_ausfahren:= ,
				b_direkttaste_ausfahren:= ,
				b_direkttaste_mittefahren:= ,
				b_direkttaste_einfahren	:= ,
				e_druckwaechter:= ST_Betriebsfreigaben.e_druckwaechter,
				i16_betriebsart:= gi16_betriebsart,
				b_no_gesteuert_im_norm_betrieb:= ,
				st_ctrl_in:= zyl_haspel_re_abspulen.st_ctrl.in,
				b_masterachse_hand_dialog_aktiv:= ,
				st_visu:= visu.st_zyl,
				st_ctrl_out=> zyl_haspel_re_abspulen.st_ctrl.out,
				a_ventil_einfahren=> ,
				a_ventil_ausfahren=> );
			
			zyl_haspel_re_sperren.fb(
				st_config:= ,
				bw_nocken_zylinder_einfahren:= ,
				bw_nocken_zylinder_ausfahren:= ,
				uw_nocken_zylinder_einfahren:= ,
				uw_nocken_zylinder_ausfahren:= ,
				b_direkttaste_ausfahren:= ,
				b_direkttaste_mittefahren:= ,
				b_direkttaste_einfahren	:= ,
				e_druckwaechter:= ST_Betriebsfreigaben.e_druckwaechter,
				i16_betriebsart:= gi16_betriebsart,
				b_no_gesteuert_im_norm_betrieb:= ,
				st_ctrl_in:= zyl_haspel_re_sperren.st_ctrl.in,
				b_masterachse_hand_dialog_aktiv:= ,
				st_visu:= visu.st_zyl,
				st_ctrl_out=> zyl_haspel_re_sperren.st_ctrl.out,
				a_ventil_einfahren=> ,
				a_ventil_ausfahren=> );
	
			zyl_bawe_halter_li.fb.st_config.b_aktiv := NOT gst_datensatz.st_md.b_wt_transport_simulation;
			zyl_bawe_halter_li.fb(
				st_config:= ,
				bw_nocken_zylinder_einfahren:= ,
				bw_nocken_zylinder_ausfahren:= ,
				uw_nocken_zylinder_einfahren:= ,
				uw_nocken_zylinder_ausfahren:= ,
				b_direkttaste_ausfahren:= ,
				b_direkttaste_mittefahren:= ,
				b_direkttaste_einfahren	:= ,
				e_druckwaechter:= ST_Betriebsfreigaben.e_druckwaechter,
				i16_betriebsart:= gi16_betriebsart,
				b_no_gesteuert_im_norm_betrieb:= ,
				st_ctrl_in:= zyl_bawe_halter_li.st_ctrl.in,
				b_masterachse_hand_dialog_aktiv:= ,
				st_visu:= visu.st_zyl,
				st_ctrl_out=> zyl_bawe_halter_li.st_ctrl.out,
				a_ventil_einfahren=> ,
				a_ventil_ausfahren=> );
	
			zyl_bawe_halter_re.fb.st_config.b_aktiv := NOT gst_datensatz.st_md.b_wt_transport_simulation;
			zyl_bawe_halter_re.fb(
				st_config:= ,
				bw_nocken_zylinder_einfahren:= ,
				bw_nocken_zylinder_ausfahren:= ,
				uw_nocken_zylinder_einfahren:= ,
				uw_nocken_zylinder_ausfahren:= ,
				b_direkttaste_ausfahren:= ,
				b_direkttaste_mittefahren:= ,
				b_direkttaste_einfahren	:= ,
				e_druckwaechter:= ST_Betriebsfreigaben.e_druckwaechter,
				i16_betriebsart:= gi16_betriebsart,
				b_no_gesteuert_im_norm_betrieb:= ,
				st_ctrl_in:= zyl_bawe_halter_re.st_ctrl.in,
				b_masterachse_hand_dialog_aktiv:= ,
				st_visu:= visu.st_zyl,
				st_ctrl_out=> zyl_bawe_halter_re.st_ctrl.out,
				a_ventil_einfahren=> ,
				a_ventil_ausfahren=> );
	
		RASTERFOLIE:
			zyl_haspel_li_heben.fb(
				st_config:= ,
				bw_nocken_zylinder_einfahren:= ,
				bw_nocken_zylinder_ausfahren:= ,
				uw_nocken_zylinder_einfahren:= ,
				uw_nocken_zylinder_ausfahren:= ,
				b_direkttaste_ausfahren:= ,
				b_direkttaste_mittefahren:= ,
				b_direkttaste_einfahren	:= ,
				e_druckwaechter:= ST_Betriebsfreigaben.e_druckwaechter,
				i16_betriebsart:= gi16_betriebsart,
				b_no_gesteuert_im_norm_betrieb:= ,
				st_ctrl_in:= zyl_haspel_li_heben.st_ctrl.in,
				b_masterachse_hand_dialog_aktiv:= ,
				st_visu:= visu.st_zyl,
				st_ctrl_out=> zyl_haspel_li_heben.st_ctrl.out,
				a_ventil_einfahren=> ,
				a_ventil_ausfahren=> );
			
			zyl_haspel_li_abspulen.fb(
				st_config:= ,
				bw_nocken_zylinder_einfahren:= ,
				bw_nocken_zylinder_ausfahren:= ,
				uw_nocken_zylinder_einfahren:= ,
				uw_nocken_zylinder_ausfahren:= ,
				b_direkttaste_ausfahren:= ,
				b_direkttaste_mittefahren:= ,
				b_direkttaste_einfahren	:= ,
				e_druckwaechter:= ST_Betriebsfreigaben.e_druckwaechter,
				i16_betriebsart:= gi16_betriebsart,
				b_no_gesteuert_im_norm_betrieb:= ,
				st_ctrl_in:= zyl_haspel_li_abspulen.st_ctrl.in,
				b_masterachse_hand_dialog_aktiv:= ,
				st_visu:= visu.st_zyl,
				st_ctrl_out=> zyl_haspel_li_abspulen.st_ctrl.out,
				a_ventil_einfahren=> ,
				a_ventil_ausfahren=> );
	
			zyl_haspel_li_sperren.fb(
				st_config:= ,
				bw_nocken_zylinder_einfahren:= ,
				bw_nocken_zylinder_ausfahren:= ,
				uw_nocken_zylinder_einfahren:= ,
				uw_nocken_zylinder_ausfahren:= ,
				b_direkttaste_ausfahren:= ,
				b_direkttaste_mittefahren:= ,
				b_direkttaste_einfahren	:= ,
				e_druckwaechter:= ST_Betriebsfreigaben.e_druckwaechter,
				i16_betriebsart:= gi16_betriebsart,
				b_no_gesteuert_im_norm_betrieb:= ,
				st_ctrl_in:= zyl_haspel_li_sperren.st_ctrl.in,
				b_masterachse_hand_dialog_aktiv:= ,
				st_visu:= visu.st_zyl,
				st_ctrl_out=> zyl_haspel_li_sperren.st_ctrl.out,
				a_ventil_einfahren=> ,
				a_ventil_ausfahren=> );
			
			zyl_haspel_re_heben.fb(
				st_config:= ,
				bw_nocken_zylinder_einfahren:= ,
				bw_nocken_zylinder_ausfahren:= ,
				uw_nocken_zylinder_einfahren:= ,
				uw_nocken_zylinder_ausfahren:= ,
				b_direkttaste_ausfahren:= ,
				b_direkttaste_mittefahren:= ,
				b_direkttaste_einfahren	:= ,
				e_druckwaechter:= ST_Betriebsfreigaben.e_druckwaechter,
				i16_betriebsart:= gi16_betriebsart,
				b_no_gesteuert_im_norm_betrieb:= ,
				st_ctrl_in:= zyl_haspel_re_heben.st_ctrl.in,
				b_masterachse_hand_dialog_aktiv:= ,
				st_visu:= visu.st_zyl,
				st_ctrl_out=> zyl_haspel_re_heben.st_ctrl.out,
				a_ventil_einfahren=> ,
				a_ventil_ausfahren=> );
			
			zyl_haspel_re_abspulen.fb(
				st_config:= ,
				bw_nocken_zylinder_einfahren:= ,
				bw_nocken_zylinder_ausfahren:= ,
				uw_nocken_zylinder_einfahren:= ,
				uw_nocken_zylinder_ausfahren:= ,
				b_direkttaste_ausfahren:= ,
				b_direkttaste_mittefahren:= ,
				b_direkttaste_einfahren	:= ,
				e_druckwaechter:= ST_Betriebsfreigaben.e_druckwaechter,
				i16_betriebsart:= gi16_betriebsart,
				b_no_gesteuert_im_norm_betrieb:= ,
				st_ctrl_in:= zyl_haspel_re_abspulen.st_ctrl.in,
				b_masterachse_hand_dialog_aktiv:= ,
				st_visu:= visu.st_zyl,
				st_ctrl_out=> zyl_haspel_re_abspulen.st_ctrl.out,
				a_ventil_einfahren=> ,
				a_ventil_ausfahren=> );
			
			zyl_haspel_re_sperren.fb(
				st_config:= ,
				bw_nocken_zylinder_einfahren:= ,
				bw_nocken_zylinder_ausfahren:= ,
				uw_nocken_zylinder_einfahren:= ,
				uw_nocken_zylinder_ausfahren:= ,
				b_direkttaste_ausfahren:= ,
				b_direkttaste_mittefahren:= ,
				b_direkttaste_einfahren	:= ,
				e_druckwaechter:= ST_Betriebsfreigaben.e_druckwaechter,
				i16_betriebsart:= gi16_betriebsart,
				b_no_gesteuert_im_norm_betrieb:= ,
				st_ctrl_in:= zyl_haspel_re_sperren.st_ctrl.in,
				b_masterachse_hand_dialog_aktiv:= ,
				st_visu:= visu.st_zyl,
				st_ctrl_out=> zyl_haspel_re_sperren.st_ctrl.out,
				a_ventil_einfahren=> ,
				a_ventil_ausfahren=> );
			
			zyl_haspel_verschieben.fb(
				st_config:= ,
				bw_nocken_zylinder_einfahren:= ,
				bw_nocken_zylinder_ausfahren:= ,
				uw_nocken_zylinder_einfahren:= ,
				uw_nocken_zylinder_ausfahren:= ,
				b_direkttaste_ausfahren:= ,
				b_direkttaste_mittefahren:= ,
				b_direkttaste_einfahren	:= ,
				e_druckwaechter:= ST_Betriebsfreigaben.e_druckwaechter,
				i16_betriebsart:= gi16_betriebsart,
				b_no_gesteuert_im_norm_betrieb:= ,
				st_ctrl_in:= zyl_haspel_verschieben.st_ctrl.in,
				b_masterachse_hand_dialog_aktiv:= ,
				st_visu:= visu.st_zyl,
				st_ctrl_out=> zyl_haspel_verschieben.st_ctrl.out,
				a_ventil_einfahren=> ,
				a_ventil_ausfahren=> );

			zyl_bandeinzuege_verschieben.fb(
				st_config:= ,
				bw_nocken_zylinder_einfahren:= ,
				bw_nocken_zylinder_ausfahren:= ,
				uw_nocken_zylinder_einfahren:= ,
				uw_nocken_zylinder_ausfahren:= ,
				b_direkttaste_ausfahren:= ,
				b_direkttaste_mittefahren:= ,
				b_direkttaste_einfahren	:= ,
				e_druckwaechter:= ST_Betriebsfreigaben.e_druckwaechter,
				i16_betriebsart:= gi16_betriebsart,
				b_no_gesteuert_im_norm_betrieb:= ,
				st_ctrl_in:= zyl_bandeinzuege_verschieben.st_ctrl.in,
				b_masterachse_hand_dialog_aktiv:= ,
				st_visu:= visu.st_zyl,
				st_ctrl_out=> zyl_bandeinzuege_verschieben.st_ctrl.out,
				a_ventil_einfahren=> ,
				a_ventil_ausfahren=> );
	
			zyl_rafo_faenger.fb.st_config.b_aktiv := NOT gst_datensatz.st_md.b_wt_transport_simulation;
			zyl_rafo_faenger.fb(
				st_config:= ,
				bw_nocken_zylinder_einfahren:= ,
				bw_nocken_zylinder_ausfahren:= ,
				uw_nocken_zylinder_einfahren:= ,
				uw_nocken_zylinder_ausfahren:= ,
				b_direkttaste_ausfahren:= ,
				b_direkttaste_mittefahren:= ,
				b_direkttaste_einfahren	:= ,
				e_druckwaechter:= ST_Betriebsfreigaben.e_druckwaechter,
				i16_betriebsart:= gi16_betriebsart,
				b_no_gesteuert_im_norm_betrieb:= ,
				st_ctrl_in:= zyl_rafo_faenger.st_ctrl.in,
				b_masterachse_hand_dialog_aktiv:= ,
				st_visu:= visu.st_zyl,
				st_ctrl_out=> zyl_rafo_faenger.st_ctrl.out,
				a_ventil_einfahren=> a_zyl_faenger_einfahren,
				a_ventil_ausfahren=> );
	
			zyl_rafo_klemmen.fb.st_config.b_aktiv := NOT gst_datensatz.st_md.b_wt_transport_simulation;
			zyl_rafo_klemmen.fb(
				st_config:= ,
				bw_nocken_zylinder_einfahren:= ,
				bw_nocken_zylinder_ausfahren:= ,
				uw_nocken_zylinder_einfahren:= ,
				uw_nocken_zylinder_ausfahren:= ,
				b_direkttaste_ausfahren:= ,
				b_direkttaste_mittefahren:= ,
				b_direkttaste_einfahren	:= ,
				e_druckwaechter:= ST_Betriebsfreigaben.e_druckwaechter,
				i16_betriebsart:= gi16_betriebsart,
				b_no_gesteuert_im_norm_betrieb:= ,
				st_ctrl_in:= zyl_rafo_klemmen.st_ctrl.in,
				b_masterachse_hand_dialog_aktiv:= ,
				st_visu:= visu.st_zyl,
				st_ctrl_out=> zyl_rafo_klemmen.st_ctrl.out,
				a_ventil_einfahren=> a_zyl_klemmen_einfahren,
				a_ventil_ausfahren=> );
	
